LIN {X 0.061,Y -334.260,Z 1455.726,A 0.000,B 0.000,C 90.000,E1 166.589} C_DIS
LIN {X 0.067,Y -335.488,Z 1455.719,A 0.000,B 0.000,C 90.000,E1 165.408} C_DIS
LIN {X 0.143,Y -340.932,Z 1455.695,A 0.000,B 0.000,C 90.000,E1 161.094} C_DIS
LIN {X -0.172,Y -342.138,Z 1455.691,A 0.000,B 0.000,C 90.000,E1 160.369} C_DIS
LIN {X 0.066,Y -342.805,Z 1455.688,A 0.000,B 0.000,C 90.000,E1 159.752} C_DIS
LIN {X 0.060,Y -429.024,Z 1455.688,A 0.000,B 0.000,C 90.000,E1 159.752} C_DIS
LIN {X -0.033,Y -430.016,Z 1455.688,A 0.000,B 0.000,C 90.000,E1 159.752} C_DIS
LIN {X 0.086,Y -433.395,Z 1455.687,A 0.000,B 0.000,C 90.000,E1 159.645} C_DIS
LIN {X -0.050,Y -435.691,Z 1455.687,A 0.000,B 0.000,C 90.000,E1 159.571} C_DIS
LIN {X -0.153,Y -438.470,Z 1455.686,A 0.000,B 0.000,C 90.000,E1 159.444} C_DIS
LIN {X -0.210,Y -444.564,Z 1455.684,A 0.000,B 0.000,C 90.000,E1 159.082} C_DIS
LIN {X 0.199,Y -450.609,Z 1455.681,A 0.000,B 0.000,C 90.000,E1 158.592} C_DIS
LIN {X 0.200,Y -458.142,Z 1455.678,A 0.000,B 0.000,C 90.000,E1 157.975} C_DIS
LIN {X 0.066,Y -470.088,Z 1455.672,A 0.000,B 0.000,C 90.000,E1 156.997} C_DIS
LIN {X 0.090,Y -477.459,Z 1455.669,A 0.000,B 0.000,C 90.000,E1 156.357} C_DIS
LIN {X -0.246,Y -486.291,Z 1455.664,A 0.000,B 0.000,C 90.000,E1 155.613} C_DIS
LIN {X -0.083,Y -496.085,Z 1455.659,A 0.000,B 0.000,C 90.000,E1 154.665} C_DIS
LIN {X -0.227,Y -500.055,Z 1455.657,A 0.000,B 0.000,C 90.000,E1 154.280} C_DIS
LIN {X 0.099,Y -504.054,Z 1455.655,A 0.000,B 0.000,C 90.000,E1 153.819} C_DIS
LIN {X -0.017,Y -509.175,Z 1455.651,A 0.000,B 0.000,C 90.000,E1 153.256} C_DIS
LIN {X -0.087,Y -512.862,Z 1455.649,A 0.000,B 0.000,C 90.000,E1 152.820} C_DIS
LIN {X -0.096,Y -517.315,Z 1455.646,A 0.000,B 0.000,C 90.000,E1 152.231} C_DIS
LIN {X -0.070,Y -521.284,Z 1455.642,A 0.000,B 0.000,C 90.000,E1 151.641} C_DIS
LIN {X -0.011,Y -524.812,Z 1455.639,A 0.000,B 0.000,C 90.000,E1 151.051} C_DIS
LIN {X 0.073,Y -528.055,Z 1455.636,A 0.000,B 0.000,C 90.000,E1 150.461} C_DIS
LIN {X 0.031,Y -531.494,Z 1455.632,A 0.000,B 0.000,C 90.000,E1 149.744} C_DIS
LIN {X 0.289,Y -534.593,Z 1455.628,A 0.000,B 0.000,C 90.000,E1 148.997} C_DIS
LIN {X -0.018,Y -536.856,Z 1455.625,A 0.000,B 0.000,C 90.000,E1 148.456} C_DIS
LIN {X 0.147,Y -538.862,Z 1455.622,A 0.000,B 0.000,C 90.000,E1 147.867} C_DIS
LIN {X -0.121,Y -541.534,Z 1455.617,A 0.000,B 0.000,C 90.000,E1 147.041} C_DIS
LIN {X 0.120,Y -544.822,Z 1455.611,A 0.000,B 0.000,C 90.000,E1 145.881} C_DIS
LIN {X -0.047,Y -547.603,Z 1455.604,A 0.000,B 0.000,C 90.000,E1 144.769} C_DIS
LIN {X 0.044,Y -548.800,Z 1455.601,A 0.000,B 0.000,C 90.000,E1 144.196} C_DIS
LIN {X 0.256,Y -550.997,Z 1455.595,A 0.000,B 0.000,C 90.000,E1 143.050} C_DIS
LIN {X -0.337,Y -552.393,Z 1455.590,A 0.000,B 0.000,C 90.000,E1 142.271} C_DIS
LIN {X 0.198,Y -553.592,Z 1455.586,A 0.000,B 0.000,C 90.000,E1 141.376} C_DIS
LIN {X 0.043,Y -554.950,Z 1455.579,A 0.000,B 0.000,C 90.000,E1 140.275} C_DIS
LIN {X -0.014,Y -556.651,Z 1455.570,A 0.000,B 0.000,C 90.000,E1 138.609} C_DIS
LIN {X -0.047,Y -558.100,Z 1455.561,A 0.000,B 0.000,C 90.000,E1 136.944} C_DIS
LIN {X 0.303,Y -559.361,Z 1455.552,A 0.000,B 0.000,C 90.000,E1 135.243} C_DIS
LIN {X 0.096,Y -559.885,Z 1455.547,A 0.000,B 0.000,C 90.000,E1 134.433} C_DIS
LIN {X 0.020,Y -560.555,Z 1455.539,A 0.000,B 0.000,C 90.000,E1 133.056} C_DIS
LIN {X 0.311,Y -560.929,Z 1455.533,A 0.000,B 0.000,C 90.000,E1 131.919} C_DIS
LIN {X -0.055,Y -561.110,Z 1455.524,A 0.000,B 0.000,C 90.000,E1 130.297} C_DIS
LIN {X -0.264,Y -561.230,Z 1455.513,A 0.000,B 0.000,C 90.000,E1 128.382} C_DIS
LIN {X -0.129,Y -561.256,Z 1455.504,A 0.000,B 0.000,C 90.000,E1 126.710} C_DIS
LIN {X -0.071,Y -561.151,Z 1455.498,A 0.000,B 0.000,C 90.000,E1 125.598} C_DIS
LIN {X 0.087,Y -560.828,Z 1455.490,A 0.000,B 0.000,C 90.000,E1 124.199} C_DIS
LIN {X -0.030,Y -560.379,Z 1455.476,A 0.000,B 0.000,C 90.000,E1 121.720} C_DIS
LIN {X -0.150,Y -560.431,Z 1455.465,A 0.000,B 0.000,C 90.000,E1 119.795} C_DIS
LIN {X -0.046,Y -560.762,Z 1455.455,A 0.000,B 0.000,C 90.000,E1 117.847} C_DIS
LIN {X 0.063,Y -561.275,Z 1455.444,A 0.000,B 0.000,C 90.000,E1 115.899} C_DIS
LIN {X -0.120,Y -561.813,Z 1455.435,A 0.000,B 0.000,C 90.000,E1 114.259} C_DIS
LIN {X -0.314,Y -562.285,Z 1455.427,A 0.000,B 0.000,C 90.000,E1 112.898} C_DIS
LIN {X 0.235,Y -562.746,Z 1455.419,A 0.000,B 0.000,C 90.000,E1 111.461} C_DIS
LIN {X -0.145,Y -563.149,Z 1455.412,A 0.000,B 0.000,C 90.000,E1 110.120} C_DIS
LIN {X 0.255,Y -563.845,Z 1455.400,A 0.000,B 0.000,C 90.000,E1 107.873} C_DIS
LIN {X -0.214,Y -564.772,Z 1455.387,A 0.000,B 0.000,C 90.000,E1 105.717} C_DIS
LIN {X -0.057,Y -564.910,Z 1455.386,A 0.000,B 0.000,C 90.000,E1 105.426} C_DIS
LIN {X 0.027,Y -565.688,Z 1455.381,A 0.000,B 0.000,C 90.000,E1 104.592} C_DIS
LIN {X 0.149,Y -566.655,Z 1455.375,A 0.000,B 0.000,C 90.000,E1 103.480} C_DIS
LIN {X 0.246,Y -567.894,Z 1455.370,A 0.000,B 0.000,C 90.000,E1 102.647} C_DIS
LIN {X -0.133,Y -568.191,Z 1455.369,A 0.000,B 0.000,C 90.000,E1 102.411} C_DIS
LIN {X 0.045,Y -569.125,Z 1455.367,A 0.000,B 0.000,C 90.000,E1 102.119} C_DIS
LIN {X 0.225,Y -569.886,Z 1455.366,A 0.000,B 0.000,C 90.000,E1 101.827} C_DIS
LIN {X 0.036,Y -569.563,Z 1455.363,A 0.000,B 0.000,C 90.000,E1 101.299} C_DIS
LIN {X 0.220,Y -569.627,Z 1455.361,A 0.000,B 0.000,C 90.000,E1 101.007} C_DIS
LIN {X 0.110,Y -569.419,Z 1455.357,A 0.000,B 0.000,C 90.000,E1 100.197} C_DIS
LIN {X -0.083,Y -569.239,Z 1455.354,A 0.000,B 0.000,C 90.000,E1 99.670} C_DIS
LIN {X 0.260,Y -568.151,Z 1455.345,A 0.000,B 0.000,C 90.000,E1 97.992} C_DIS
LIN {X -0.248,Y -568.138,Z 1455.339,A 0.000,B 0.000,C 90.000,E1 96.947} C_DIS
LIN {X -0.202,Y -570.184,Z 1455.319,A 0.000,B 0.000,C 90.000,E1 93.383} C_DIS
LIN {X 0.188,Y -571.720,Z 1455.308,A 0.000,B 0.000,C 90.000,E1 91.432} C_DIS
LIN {X -0.131,Y -573.048,Z 1455.299,A 0.000,B 0.000,C 90.000,E1 89.828} C_DIS
LIN {X 0.005,Y -574.147,Z 1455.292,A 0.000,B 0.000,C 90.000,E1 88.453} C_DIS
LIN {X 0.028,Y -575.123,Z 1455.285,A 0.000,B 0.000,C 90.000,E1 87.364} C_DIS
LIN {X 0.213,Y -576.306,Z 1455.278,A 0.000,B 0.000,C 90.000,E1 85.988} C_DIS
LIN {X 0.222,Y -577.984,Z 1455.267,A 0.000,B 0.000,C 90.000,E1 84.090} C_DIS
LIN {X 0.197,Y -579.406,Z 1455.258,A 0.000,B 0.000,C 90.000,E1 82.470} C_DIS
LIN {X 0.211,Y -580.977,Z 1455.249,A 0.000,B 0.000,C 90.000,E1 80.849} C_DIS
LIN {X -0.222,Y -582.503,Z 1455.240,A 0.000,B 0.000,C 90.000,E1 79.275} C_DIS
LIN {X -0.295,Y -583.830,Z 1455.233,A 0.000,B 0.000,C 90.000,E1 77.937} C_DIS
LIN {X -0.236,Y -585.030,Z 1455.225,A 0.000,B 0.000,C 90.000,E1 76.589} C_DIS
LIN {X 0.222,Y -586.205,Z 1455.216,A 0.000,B 0.000,C 90.000,E1 74.936} C_DIS
LIN {X -0.027,Y -586.651,Z 1455.212,A 0.000,B 0.000,C 90.000,E1 74.157} C_DIS
LIN {X 0.058,Y -587.614,Z 1455.203,A 0.000,B 0.000,C 90.000,E1 72.543} C_DIS
LIN {X -0.083,Y -588.287,Z 1455.196,A 0.000,B 0.000,C 90.000,E1 71.221} C_DIS
LIN {X -0.021,Y -589.004,Z 1455.188,A 0.000,B 0.000,C 90.000,E1 69.880} C_DIS
LIN {X -0.180,Y -590.083,Z 1455.178,A 0.000,B 0.000,C 90.000,E1 68.028} C_DIS
LIN {X 0.026,Y -590.928,Z 1455.169,A 0.000,B 0.000,C 90.000,E1 66.410} C_DIS
LIN {X 0.039,Y -592.327,Z 1455.157,A 0.000,B 0.000,C 90.000,E1 64.280} C_DIS
LIN {X 0.177,Y -593.164,Z 1455.151,A 0.000,B 0.000,C 90.000,E1 63.204} C_DIS
LIN {X -0.300,Y -595.310,Z 1455.135,A 0.000,B 0.000,C 90.000,E1 60.333} C_DIS
LIN {X -0.071,Y -596.270,Z 1455.129,A 0.000,B 0.000,C 90.000,E1 59.253} C_DIS
LIN {X 0.219,Y -597.873,Z 1455.119,A 0.000,B 0.000,C 90.000,E1 57.375} C_DIS
LIN {X 0.026,Y -599.521,Z 1455.109,A 0.000,B 0.000,C 90.000,E1 55.548} C_DIS
LIN {X -0.197,Y -600.841,Z 1455.100,A 0.000,B 0.000,C 90.000,E1 53.989} C_DIS
LIN {X -0.028,Y -601.825,Z 1455.091,A 0.000,B 0.000,C 90.000,E1 52.396} C_DIS
LIN {X -0.087,Y -602.718,Z 1455.084,A 0.000,B 0.000,C 90.000,E1 51.090} C_DIS
LIN {X 0.205,Y -603.243,Z 1455.079,A 0.000,B 0.000,C 90.000,E1 50.275} C_DIS
LIN {X 0.247,Y -603.524,Z 1455.077,A 0.000,B 0.000,C 90.000,E1 49.747} C_DIS
LIN {X 0.135,Y -603.708,Z 1455.069,A 0.000,B 0.000,C 90.000,E1 48.447} C_DIS
LIN {X 0.026,Y -603.994,Z 1455.062,A 0.000,B 0.000,C 90.000,E1 47.148} C_DIS
LIN {X 0.327,Y -604.187,Z 1455.055,A 0.000,B 0.000,C 90.000,E1 45.810} C_DIS
LIN {X -0.036,Y -604.000,Z 1455.049,A 0.000,B 0.000,C 90.000,E1 44.798} C_DIS
LIN {X 0.036,Y -603.534,Z 1455.043,A 0.000,B 0.000,C 90.000,E1 43.743} C_DIS
LIN {X 0.089,Y -602.845,Z 1455.037,A 0.000,B 0.000,C 90.000,E1 42.690} C_DIS
LIN {X -0.076,Y -602.179,Z 1455.033,A 0.000,B 0.000,C 90.000,E1 41.919} C_DIS
LIN {X -0.219,Y -600.878,Z 1455.026,A 0.000,B 0.000,C 90.000,E1 40.620} C_DIS
LIN {X 0.072,Y -599.204,Z 1455.018,A 0.000,B 0.000,C 90.000,E1 39.277} C_DIS
LIN {X -0.042,Y -597.395,Z 1455.011,A 0.000,B 0.000,C 90.000,E1 37.971} C_DIS
LIN {X -0.059,Y -595.733,Z 1455.005,A 0.000,B 0.000,C 90.000,E1 36.916} C_DIS
LIN {X 0.010,Y -593.691,Z 1454.999,A 0.000,B 0.000,C 90.000,E1 35.851} C_DIS
LIN {X 0.318,Y -591.888,Z 1454.995,A 0.000,B 0.000,C 90.000,E1 35.025} C_DIS
LIN {X 0.126,Y -589.909,Z 1454.990,A 0.000,B 0.000,C 90.000,E1 34.246} C_DIS
LIN {X 0.073,Y -587.854,Z 1454.986,A 0.000,B 0.000,C 90.000,E1 33.452} C_DIS
LIN {X -0.166,Y -585.459,Z 1454.981,A 0.000,B 0.000,C 90.000,E1 32.673} C_DIS
LIN {X -0.082,Y -581.947,Z 1454.975,A 0.000,B 0.000,C 90.000,E1 31.592} C_DIS
LIN {X -0.060,Y -579.976,Z 1454.973,A 0.000,B 0.000,C 90.000,E1 31.052} C_DIS
LIN {X -0.201,Y -576.507,Z 1454.968,A 0.000,B 0.000,C 90.000,E1 30.256} C_DIS
LIN {X 0.201,Y -573.334,Z 1454.964,A 0.000,B 0.000,C 90.000,E1 29.539} C_DIS
LIN {X -0.100,Y -568.447,Z 1454.959,A 0.000,B 0.000,C 90.000,E1 28.615} C_DIS
LIN {X 0.221,Y -564.672,Z 1454.955,A 0.000,B 0.000,C 90.000,E1 27.897} C_DIS
LIN {X 0.149,Y -559.808,Z 1454.951,A 0.000,B 0.000,C 90.000,E1 27.078} C_DIS
LIN {X 0.282,Y -554.507,Z 1454.946,A 0.000,B 0.000,C 90.000,E1 26.232} C_DIS
LIN {X -0.158,Y -550.742,Z 1454.943,A 0.000,B 0.000,C 90.000,E1 25.720} C_DIS
LIN {X -0.005,Y -547.790,Z 1454.941,A 0.000,B 0.000,C 90.000,E1 25.283} C_DIS
LIN {X 0.121,Y -540.180,Z 1454.935,A 0.000,B 0.000,C 90.000,E1 24.283} C_DIS
LIN {X -0.054,Y -534.418,Z 1454.931,A 0.000,B 0.000,C 90.000,E1 23.590} C_DIS
LIN {X -0.009,Y -525.864,Z 1454.926,A 0.000,B 0.000,C 90.000,E1 22.589} C_DIS
LIN {X -0.101,Y -520.741,Z 1454.922,A 0.000,B 0.000,C 90.000,E1 22.025} C_DIS
LIN {X -0.243,Y -511.542,Z 1454.917,A 0.000,B 0.000,C 90.000,E1 21.046} C_DIS
LIN {X 0.088,Y -500.576,Z 1454.911,A 0.000,B 0.000,C 90.000,E1 19.885} C_DIS
LIN {X 0.019,Y -492.405,Z 1454.906,A 0.000,B 0.000,C 90.000,E1 19.087} C_DIS
LIN {X 0.151,Y -487.808,Z 1454.904,A 0.000,B 0.000,C 90.000,E1 18.671} C_DIS
LIN {X 0.072,Y -482.816,Z 1454.902,A 0.000,B 0.000,C 90.000,E1 18.308} C_DIS
LIN {X -0.111,Y -479.110,Z 1454.901,A 0.000,B 0.000,C 90.000,E1 18.109} C_DIS
LIN {X -0.157,Y -476.473,Z 1454.900,A 0.000,B 0.000,C 90.000,E1 18.000} C_DIS
LIN {X -0.126,Y -474.326,Z 1454.900,A 0.000,B 0.000,C 90.000,E1 17.946} C_DIS
LIN {X -0.156,Y -473.854,Z 1454.900,A 0.000,B 0.000,C 90.000,E1 17.946} C_DIS
LIN {X -0.147,Y -373.992,Z 1454.900,A 0.000,B 0.000,C 90.000,E1 17.946} C_DIS
LIN {X 0.091,Y -373.673,Z 1454.897,A 0.000,B 0.000,C 90.000,E1 17.528} C_DIS
LIN {X -0.129,Y -368.069,Z 1454.869,A 0.000,B 0.000,C 90.000,E1 12.411} C_DIS
LIN {X 0.039,Y -366.383,Z 1454.854,A 0.000,B 0.000,C 90.000,E1 9.792} C_DIS
LIN {X -0.021,Y -361.732,Z 1454.821,A 0.000,B 0.000,C 90.000,E1 3.841} C_DIS
LIN {X -0.136,Y -360.851,Z 1454.801,A 0.000,B 0.000,C 90.000,E1 0.115} C_DIS
LIN {X -0.053,Y -359.426,Z 1454.770,A 0.000,B 0.000,C 90.000,E1 354.546} C_DIS
LIN {X 0.070,Y -358.890,Z 1454.759,A 0.000,B 0.000,C 90.000,E1 352.648} C_DIS
LIN {X -0.020,Y -359.563,Z 1454.726,A 0.000,B 0.000,C 90.000,E1 346.645} C_DIS
LIN {X 0.001,Y -361.801,Z 1454.684,A 0.000,B 0.000,C 90.000,E1 339.135} C_DIS
LIN {X -0.154,Y -362.053,Z 1454.680,A 0.000,B 0.000,C 90.000,E1 338.411} C_DIS
LIN {X 0.189,Y -365.980,Z 1454.643,A 0.000,B 0.000,C 90.000,E1 331.641} C_DIS
LIN {X 0.029,Y -366.387,Z 1454.639,A 0.000,B 0.000,C 90.000,E1 330.923} C_DIS
LIN {X -0.031,Y -371.355,Z 1454.604,A 0.000,B 0.000,C 90.000,E1 324.642} C_DIS
LIN {X -0.043,Y -371.766,Z 1454.602,A 0.000,B 0.000,C 90.000,E1 324.276} C_DIS
LIN {X 0.013,Y -377.358,Z 1454.567,A 0.000,B 0.000,C 90.000,E1 318.038} C_DIS
LIN {X 0.012,Y -378.235,Z 1454.563,A 0.000,B 0.000,C 90.000,E1 317.310} C_DIS
LIN {X 0.002,Y -383.940,Z 1454.531,A 0.000,B 0.000,C 90.000,E1 311.515} C_DIS
LIN {X 0.088,Y -384.893,Z 1454.527,A 0.000,B 0.000,C 90.000,E1 310.782} C_DIS
LIN {X 0.262,Y -390.610,Z 1454.495,A 0.000,B 0.000,C 90.000,E1 305.025} C_DIS
LIN {X 0.106,Y -391.104,Z 1454.493,A 0.000,B 0.000,C 90.000,E1 304.692} C_DIS
LIN {X 0.022,Y -391.648,Z 1454.489,A 0.000,B 0.000,C 90.000,E1 303.992} C_DIS
LIN {X -0.080,Y -396.825,Z 1454.459,A 0.000,B 0.000,C 90.000,E1 298.693} C_DIS
LIN {X -0.210,Y -397.120,Z 1454.457,A 0.000,B 0.000,C 90.000,E1 298.359} C_DIS
LIN {X -0.055,Y -401.597,Z 1454.426,A 0.000,B 0.000,C 90.000,E1 292.717} C_DIS
LIN {X 0.222,Y -404.659,Z 1454.395,A 0.000,B 0.000,C 90.000,E1 287.094} C_DIS
LIN {X -0.079,Y -404.735,Z 1454.391,A 0.000,B 0.000,C 90.000,E1 286.441} C_DIS
LIN {X 0.214,Y -406.099,Z 1454.364,A 0.000,B 0.000,C 90.000,E1 281.535} C_DIS
LIN {X -0.176,Y -406.094,Z 1454.362,A 0.000,B 0.000,C 90.000,E1 281.243} C_DIS
LIN {X -0.097,Y -405.680,Z 1454.333,A 0.000,B 0.000,C 90.000,E1 276.024} C_DIS
LIN {X -0.165,Y -405.058,Z 1454.328,A 0.000,B 0.000,C 90.000,E1 274.992} C_DIS
LIN {X -0.060,Y -403.497,Z 1454.304,A 0.000,B 0.000,C 90.000,E1 270.802} C_DIS
LIN {X -0.092,Y -403.288,Z 1454.302,A 0.000,B 0.000,C 90.000,E1 270.458} C_DIS
LIN {X 0.091,Y -398.931,Z 1454.271,A 0.000,B 0.000,C 90.000,E1 264.837} C_DIS
LIN {X -0.040,Y -393.108,Z 1454.242,A 0.000,B 0.000,C 90.000,E1 259.567} C_DIS
LIN {X -0.079,Y -392.835,Z 1454.240,A 0.000,B 0.000,C 90.000,E1 259.218} C_DIS
LIN {X 0.034,Y -385.993,Z 1454.212,A 0.000,B 0.000,C 90.000,E1 254.212} C_DIS
LIN {X -0.026,Y -385.267,Z 1454.208,A 0.000,B 0.000,C 90.000,E1 253.504} C_DIS
LIN {X -0.004,Y -384.768,Z 1454.206,A 0.000,B 0.000,C 90.000,E1 253.142} C_DIS
LIN {X 0.221,Y -377.973,Z 1454.182,A 0.000,B 0.000,C 90.000,E1 248.773} C_DIS
LIN {X -0.044,Y -376.233,Z 1454.174,A 0.000,B 0.000,C 90.000,E1 247.358} C_DIS
LIN {X 0.057,Y -374.944,Z 1454.170,A 0.000,B 0.000,C 90.000,E1 246.613} C_DIS
LIN {X -0.208,Y -368.417,Z 1454.148,A 0.000,B 0.000,C 90.000,E1 242.615} C_DIS
LIN {X 0.097,Y -366.047,Z 1454.137,A 0.000,B 0.000,C 90.000,E1 240.717} C_DIS
LIN {X 0.004,Y -359.196,Z 1454.115,A 0.000,B 0.000,C 90.000,E1 236.628} C_DIS
LIN {X 0.021,Y -355.842,Z 1454.100,A 0.000,B 0.000,C 90.000,E1 233.989} C_DIS
LIN {X -0.173,Y -348.793,Z 1454.075,A 0.000,B 0.000,C 90.000,E1 229.461} C_DIS
LIN {X -0.097,Y -346.185,Z 1454.062,A 0.000,B 0.000,C 90.000,E1 227.148} C_DIS
LIN {X -0.088,Y -345.065,Z 1454.058,A 0.000,B 0.000,C 90.000,E1 226.377} C_DIS
LIN {X 0.094,Y -338.586,Z 1454.030,A 0.000,B 0.000,C 90.000,E1 221.310} C_DIS
LIN {X 0.094,Y -336.840,Z 1454.019,A 0.000,B 0.000,C 90.000,E1 219.358} C_DIS
LIN {X 0.014,Y -330.861,Z 1453.988,A 0.000,B 0.000,C 90.000,E1 213.865} C_DIS
LIN {X 0.149,Y -329.296,Z 1453.975,A 0.000,B 0.000,C 90.000,E1 211.465} C_DIS
LIN {X -0.154,Y -324.669,Z 1453.942,A 0.000,B 0.000,C 90.000,E1 205.540} C_DIS
LIN {X 0.174,Y -323.837,Z 1453.928,A 0.000,B 0.000,C 90.000,E1 203.078} C_DIS
LIN {X -0.017,Y -321.124,Z 1453.881,A 0.000,B 0.000,C 90.000,E1 194.662} C_DIS
LIN {X 0.138,Y -320.932,Z 1453.877,A 0.000,B 0.000,C 90.000,E1 193.828} C_DIS
LIN {X -0.076,Y -321.562,Z 1453.832,A 0.000,B 0.000,C 90.000,E1 185.796} C_DIS
LIN {X -0.143,Y -324.415,Z 1453.790,A 0.000,B 0.000,C 90.000,E1 178.165} C_DIS
LIN {X -0.141,Y -325.376,Z 1453.783,A 0.000,B 0.000,C 90.000,E1 176.963} C_DIS
LIN {X -0.100,Y -329.112,Z 1453.750,A 0.000,B 0.000,C 90.000,E1 170.971} C_DIS
LIN {X 0.061,Y -334.260,Z 1453.726,A 0.000,B 0.000,C 90.000,E1 166.589} C_DIS
LIN {X 0.067,Y -335.488,Z 1453.719,A 0.000,B 0.000,C 90.000,E1 165.408} C_DIS
LIN {X 0.143,Y -340.932,Z 1453.695,A 0.000,B 0.000,C 90.000,E1 161.094} C_DIS
LIN {X 0.033,Y -342.089,Z 1453.691,A 0.000,B 0.000,C 90.000,E1 160.369} C_DIS
LIN {X 0.017,Y -422.192,Z 1453.691,A 0.000,B 0.000,C 90.000,E1 160.369} C_DIS
LIN {X -0.214,Y -424.388,Z 1453.691,A 0.000,B 0.000,C 90.000,E1 160.369} C_DIS
LIN {X -0.104,Y -426.356,Z 1453.691,A 0.000,B 0.000,C 90.000,E1 160.296} C_DIS
LIN {X -0.097,Y -429.003,Z 1453.690,A 0.000,B 0.000,C 90.000,E1 160.188} C_DIS
LIN {X -0.214,Y -431.860,Z 1453.689,A 0.000,B 0.000,C 90.000,E1 160.061} C_DIS
LIN {X -0.149,Y -434.914,Z 1453.688,A 0.000,B 0.000,C 90.000,E1 159.880} C_DIS
LIN {X -0.230,Y -437.978,Z 1453.687,A 0.000,B 0.000,C 90.000,E1 159.699} C_DIS
LIN {X 0.171,Y -444.013,Z 1453.685,A 0.000,B 0.000,C 90.000,E1 159.209} C_DIS
LIN {X 0.148,Y -450.072,Z 1453.682,A 0.000,B 0.000,C 90.000,E1 158.720} C_DIS
LIN {X -0.045,Y -465.121,Z 1453.675,A 0.000,B 0.000,C 90.000,E1 157.486} C_DIS
LIN {X -0.224,Y -475.642,Z 1453.670,A 0.000,B 0.000,C 90.000,E1 156.613} C_DIS
LIN {X 0.111,Y -484.431,Z 1453.666,A 0.000,B 0.000,C 90.000,E1 155.793} C_DIS
LIN {X -0.122,Y -491.613,Z 1453.662,A 0.000,B 0.000,C 90.000,E1 155.153} C_DIS
LIN {X 0.108,Y -498.531,Z 1453.658,A 0.000,B 0.000,C 90.000,E1 154.460} C_DIS
LIN {X 0.007,Y -505.152,Z 1453.654,A 0.000,B 0.000,C 90.000,E1 153.768} C_DIS
LIN {X 0.016,Y -509.028,Z 1453.652,A 0.000,B 0.000,C 90.000,E1 153.332} C_DIS
LIN {X 0.016,Y -513.849,Z 1453.649,A 0.000,B 0.000,C 90.000,E1 152.743} C_DIS
LIN {X 0.188,Y -517.252,Z 1453.646,A 0.000,B 0.000,C 90.000,E1 152.281} C_DIS
LIN {X -0.029,Y -521.248,Z 1453.643,A 0.000,B 0.000,C 90.000,E1 151.719} C_DIS
LIN {X -0.133,Y -525.606,Z 1453.639,A 0.000,B 0.000,C 90.000,E1 151.001} C_DIS
LIN {X 0.109,Y -528.058,Z 1453.636,A 0.000,B 0.000,C 90.000,E1 150.539} C_DIS
LIN {X 0.065,Y -531.547,Z 1453.632,A 0.000,B 0.000,C 90.000,E1 149.822} C_DIS
LIN {X -0.138,Y -534.673,Z 1453.628,A 0.000,B 0.000,C 90.000,E1 149.125} C_DIS
LIN {X 0.015,Y -536.937,Z 1453.625,A 0.000,B 0.000,C 90.000,E1 148.535} C_DIS
LIN {X -0.277,Y -538.954,Z 1453.622,A 0.000,B 0.000,C 90.000,E1 147.995} C_DIS
LIN {X -0.090,Y -541.642,Z 1453.617,A 0.000,B 0.000,C 90.000,E1 147.120} C_DIS
LIN {X 0.149,Y -544.927,Z 1453.611,A 0.000,B 0.000,C 90.000,E1 145.960} C_DIS
LIN {X -0.018,Y -547.714,Z 1453.605,A 0.000,B 0.000,C 90.000,E1 144.848} C_DIS
LIN {X 0.071,Y -548.928,Z 1453.602,A 0.000,B 0.000,C 90.000,E1 144.276} C_DIS
LIN {X 0.284,Y -551.125,Z 1453.595,A 0.000,B 0.000,C 90.000,E1 143.130} C_DIS
LIN {X 0.092,Y -552.923,Z 1453.589,A 0.000,B 0.000,C 90.000,E1 142.029} C_DIS
LIN {X 0.293,Y -554.055,Z 1453.584,A 0.000,B 0.000,C 90.000,E1 141.170} C_DIS
LIN {X 0.140,Y -555.357,Z 1453.578,A 0.000,B 0.000,C 90.000,E1 140.070} C_DIS
LIN {X 0.012,Y -556.744,Z 1453.571,A 0.000,B 0.000,C 90.000,E1 138.690} C_DIS
LIN {X -0.018,Y -558.172,Z 1453.561,A 0.000,B 0.000,C 90.000,E1 137.025} C_DIS
LIN {X -0.061,Y -559.419,Z 1453.552,A 0.000,B 0.000,C 90.000,E1 135.364} C_DIS
LIN {X -0.205,Y -560.071,Z 1453.546,A 0.000,B 0.000,C 90.000,E1 134.271} C_DIS
LIN {X 0.131,Y -560.719,Z 1453.538,A 0.000,B 0.000,C 90.000,E1 132.852} C_DIS
LIN {X 0.013,Y -561.021,Z 1453.532,A 0.000,B 0.000,C 90.000,E1 131.757} C_DIS
LIN {X 0.072,Y -561.165,Z 1453.523,A 0.000,B 0.000,C 90.000,E1 130.092} C_DIS
LIN {X -0.130,Y -561.245,Z 1453.512,A 0.000,B 0.000,C 90.000,E1 128.177} C_DIS
LIN {X 0.010,Y -561.246,Z 1453.503,A 0.000,B 0.000,C 90.000,E1 126.503} C_DIS
LIN {X 0.070,Y -561.093,Z 1453.497,A 0.000,B 0.000,C 90.000,E1 125.391} C_DIS
LIN {X 0.134,Y -560.851,Z 1453.491,A 0.000,B 0.000,C 90.000,E1 124.278} C_DIS
LIN {X 0.025,Y -560.386,Z 1453.477,A 0.000,B 0.000,C 90.000,E1 121.799} C_DIS
LIN {X -0.088,Y -560.401,Z 1453.466,A 0.000,B 0.000,C 90.000,E1 119.873} C_DIS
LIN {X 0.284,Y -560.752,Z 1453.455,A 0.000,B 0.000,C 90.000,E1 117.897} C_DIS
LIN {X 0.138,Y -561.251,Z 1453.444,A 0.000,B 0.000,C 90.000,E1 115.976} C_DIS
LIN {X -0.037,Y -561.811,Z 1453.435,A 0.000,B 0.000,C 90.000,E1 114.335} C_DIS
LIN {X -0.006,Y -562.287,Z 1453.427,A 0.000,B 0.000,C 90.000,E1 112.950} C_DIS
LIN {X -0.191,Y -562.759,Z 1453.420,A 0.000,B 0.000,C 90.000,E1 111.589} C_DIS
LIN {X 0.154,Y -563.162,Z 1453.412,A 0.000,B 0.000,C 90.000,E1 110.174} C_DIS
LIN {X 0.155,Y -563.984,Z 1453.398,A 0.000,B 0.000,C 90.000,E1 107.692} C_DIS
LIN {X -0.161,Y -564.613,Z 1453.392,A 0.000,B 0.000,C 90.000,E1 106.622} C_DIS
LIN {X -0.235,Y -565.155,Z 1453.389,A 0.000,B 0.000,C 90.000,E1 106.079} C_DIS
LIN {X 0.236,Y -565.472,Z 1453.386,A 0.000,B 0.000,C 90.000,E1 105.481} C_DIS
LIN {X 0.033,Y -565.836,Z 1453.385,A 0.000,B 0.000,C 90.000,E1 105.300} C_DIS
LIN {X 0.151,Y -566.728,Z 1453.381,A 0.000,B 0.000,C 90.000,E1 104.481} C_DIS
LIN {X 0.108,Y -566.741,Z 1453.381,A 0.000,B 0.000,C 90.000,E1 104.481} C_DIS
LIN {X 0.085,Y -568.453,Z 1453.376,A 0.000,B 0.000,C 90.000,E1 103.647} C_DIS
LIN {X 0.261,Y -568.762,Z 1453.374,A 0.000,B 0.000,C 90.000,E1 103.355} C_DIS
LIN {X 0.253,Y -570.843,Z 1453.370,A 0.000,B 0.000,C 90.000,E1 102.535} C_DIS
LIN {X -0.117,Y -571.767,Z 1453.368,A 0.000,B 0.000,C 90.000,E1 102.299} C_DIS
LIN {X -0.051,Y -572.232,Z 1453.366,A 0.000,B 0.000,C 90.000,E1 101.883} C_DIS
LIN {X 0.267,Y -572.517,Z 1453.365,A 0.000,B 0.000,C 90.000,E1 101.715} C_DIS
LIN {X 0.099,Y -572.809,Z 1453.362,A 0.000,B 0.000,C 90.000,E1 101.186} C_DIS
LIN {X -0.266,Y -572.851,Z 1453.361,A 0.000,B 0.000,C 90.000,E1 100.950} C_DIS
LIN {X -0.070,Y -572.533,Z 1453.359,A 0.000,B 0.000,C 90.000,E1 100.658} C_DIS
LIN {X 0.127,Y -572.455,Z 1453.358,A 0.000,B 0.000,C 90.000,E1 100.366} C_DIS
LIN {X 0.221,Y -571.945,Z 1453.356,A 0.000,B 0.000,C 90.000,E1 100.084} C_DIS
LIN {X 0.047,Y -571.563,Z 1453.353,A 0.000,B 0.000,C 90.000,E1 99.557} C_DIS
LIN {X -0.034,Y -570.180,Z 1453.349,A 0.000,B 0.000,C 90.000,E1 98.746} C_DIS
LIN {X 0.152,Y -569.572,Z 1453.347,A 0.000,B 0.000,C 90.000,E1 98.454} C_DIS
LIN {X 0.104,Y -568.992,Z 1453.345,A 0.000,B 0.000,C 90.000,E1 98.049} C_DIS
LIN {X -0.162,Y -568.709,Z 1453.342,A 0.000,B 0.000,C 90.000,E1 97.530} C_DIS
LIN {X 0.015,Y -568.756,Z 1453.340,A 0.000,B 0.000,C 90.000,E1 97.239} C_DIS
LIN {X -0.271,Y -568.501,Z 1453.337,A 0.000,B 0.000,C 90.000,E1 96.720} C_DIS
LIN {X 0.283,Y -569.347,Z 1453.325,A 0.000,B 0.000,C 90.000,E1 94.473} C_DIS
LIN {X 0.085,Y -570.814,Z 1453.314,A 0.000,B 0.000,C 90.000,E1 92.579} C_DIS
LIN {X -0.240,Y -572.162,Z 1453.305,A 0.000,B 0.000,C 90.000,E1 90.974} C_DIS
LIN {X 0.166,Y -573.729,Z 1453.295,A 0.000,B 0.000,C 90.000,E1 89.026} C_DIS
LIN {X -0.099,Y -575.147,Z 1453.286,A 0.000,B 0.000,C 90.000,E1 87.421} C_DIS
LIN {X 0.273,Y -576.558,Z 1453.277,A 0.000,B 0.000,C 90.000,E1 85.755} C_DIS
LIN {X 0.302,Y -578.263,Z 1453.266,A 0.000,B 0.000,C 90.000,E1 83.856} C_DIS
LIN {X 0.214,Y -579.710,Z 1453.257,A 0.000,B 0.000,C 90.000,E1 82.243} C_DIS
LIN {X 0.092,Y -581.050,Z 1453.250,A 0.000,B 0.000,C 90.000,E1 80.905} C_DIS
LIN {X 0.128,Y -582.583,Z 1453.241,A 0.000,B 0.000,C 90.000,E1 79.285} C_DIS
LIN {X 0.165,Y -583.939,Z 1453.233,A 0.000,B 0.000,C 90.000,E1 77.937} C_DIS
LIN {X 0.227,Y -585.128,Z 1453.226,A 0.000,B 0.000,C 90.000,E1 76.589} C_DIS
LIN {X -0.121,Y -586.121,Z 1453.218,A 0.000,B 0.000,C 90.000,E1 75.283} C_DIS
LIN {X -0.125,Y -586.786,Z 1453.212,A 0.000,B 0.000,C 90.000,E1 74.212} C_DIS
LIN {X -0.033,Y -587.735,Z 1453.203,A 0.000,B 0.000,C 90.000,E1 72.598} C_DIS
LIN {X -0.167,Y -588.408,Z 1453.196,A 0.000,B 0.000,C 90.000,E1 71.275} C_DIS
LIN {X -0.098,Y -589.135,Z 1453.188,A 0.000,B 0.000,C 90.000,E1 69.934} C_DIS
LIN {X 0.079,Y -590.192,Z 1453.178,A 0.000,B 0.000,C 90.000,E1 68.050} C_DIS
LIN {X -0.270,Y -591.053,Z 1453.169,A 0.000,B 0.000,C 90.000,E1 66.485} C_DIS
LIN {X -0.106,Y -592.640,Z 1453.156,A 0.000,B 0.000,C 90.000,E1 64.076} C_DIS
LIN {X 0.042,Y -593.409,Z 1453.150,A 0.000,B 0.000,C 90.000,E1 62.999} C_DIS
LIN {X 0.195,Y -595.442,Z 1453.135,A 0.000,B 0.000,C 90.000,E1 60.333} C_DIS
LIN {X 0.335,Y -596.590,Z 1453.128,A 0.000,B 0.000,C 90.000,E1 58.997} C_DIS
LIN {X -0.105,Y -597.984,Z 1453.119,A 0.000,B 0.000,C 90.000,E1 57.454} C_DIS
LIN {X -0.201,Y -599.385,Z 1453.110,A 0.000,B 0.000,C 90.000,E1 55.881} C_DIS
LIN {X 0.176,Y -600.083,Z 1453.106,A 0.000,B 0.000,C 90.000,E1 55.055} C_DIS
LIN {X -0.280,Y -601.167,Z 1453.099,A 0.000,B 0.000,C 90.000,E1 53.783} C_DIS
LIN {X 0.145,Y -602.380,Z 1453.089,A 0.000,B 0.000,C 90.000,E1 51.904} C_DIS
LIN {X 0.086,Y -603.252,Z 1453.081,A 0.000,B 0.000,C 90.000,E1 50.598} C_DIS
LIN {X 0.169,Y -603.773,Z 1453.075,A 0.000,B 0.000,C 90.000,E1 49.542} C_DIS
LIN {X 0.100,Y -604.075,Z 1453.065,A 0.000,B 0.000,C 90.000,E1 47.715} C_DIS
LIN {X 0.200,Y -604.388,Z 1453.057,A 0.000,B 0.000,C 90.000,E1 46.134} C_DIS
LIN {X 0.267,Y -604.288,Z 1453.051,A 0.000,B 0.000,C 90.000,E1 45.081} C_DIS
LIN {X -0.323,Y -604.032,Z 1453.046,A 0.000,B 0.000,C 90.000,E1 44.352} C_DIS
LIN {X -0.024,Y -603.283,Z 1453.039,A 0.000,B 0.000,C 90.000,E1 43.014} C_DIS
LIN {X 0.016,Y -602.465,Z 1453.033,A 0.000,B 0.000,C 90.000,E1 41.962} C_DIS
LIN {X 0.325,Y -601.194,Z 1453.026,A 0.000,B 0.000,C 90.000,E1 40.620} C_DIS
LIN {X -0.225,Y -599.549,Z 1453.019,A 0.000,B 0.000,C 90.000,E1 39.358} C_DIS
LIN {X 0.038,Y -597.733,Z 1453.011,A 0.000,B 0.000,C 90.000,E1 38.016} C_DIS
LIN {X 0.139,Y -596.110,Z 1453.005,A 0.000,B 0.000,C 90.000,E1 36.950} C_DIS
LIN {X 0.220,Y -594.085,Z 1453.000,A 0.000,B 0.000,C 90.000,E1 35.884} C_DIS
LIN {X 0.270,Y -591.676,Z 1452.994,A 0.000,B 0.000,C 90.000,E1 34.818} C_DIS
LIN {X -0.052,Y -589.005,Z 1452.988,A 0.000,B 0.000,C 90.000,E1 33.785} C_DIS
LIN {X 0.214,Y -586.766,Z 1452.983,A 0.000,B 0.000,C 90.000,E1 32.959} C_DIS
LIN {X -0.177,Y -583.400,Z 1452.977,A 0.000,B 0.000,C 90.000,E1 31.926} C_DIS
LIN {X -0.145,Y -581.551,Z 1452.974,A 0.000,B 0.000,C 90.000,E1 31.386} C_DIS
LIN {X -0.125,Y -579.525,Z 1452.971,A 0.000,B 0.000,C 90.000,E1 30.846} C_DIS
LIN {X 0.302,Y -576.554,Z 1452.968,A 0.000,B 0.000,C 90.000,E1 30.129} C_DIS
LIN {X 0.203,Y -573.396,Z 1452.964,A 0.000,B 0.000,C 90.000,E1 29.461} C_DIS
LIN {X -0.288,Y -569.188,Z 1452.959,A 0.000,B 0.000,C 90.000,E1 28.693} C_DIS
LIN {X -0.046,Y -564.674,Z 1452.955,A 0.000,B 0.000,C 90.000,E1 27.847} C_DIS
LIN {X 0.143,Y -559.815,Z 1452.950,A 0.000,B 0.000,C 90.000,E1 27.001} C_DIS
LIN {X 0.027,Y -554.512,Z 1452.946,A 0.000,B 0.000,C 90.000,E1 26.181} C_DIS
LIN {X 0.211,Y -549.757,Z 1452.942,A 0.000,B 0.000,C 90.000,E1 25.463} C_DIS
LIN {X 0.235,Y -545.611,Z 1452.938,A 0.000,B 0.000,C 90.000,E1 24.899} C_DIS
LIN {X -0.023,Y -539.009,Z 1452.934,A 0.000,B 0.000,C 90.000,E1 24.079} C_DIS
LIN {X -0.072,Y -534.355,Z 1452.931,A 0.000,B 0.000,C 90.000,E1 23.515} C_DIS
LIN {X -0.044,Y -525.756,Z 1452.925,A 0.000,B 0.000,C 90.000,E1 22.514} C_DIS
LIN {X 0.195,Y -519.315,Z 1452.921,A 0.000,B 0.000,C 90.000,E1 21.770} C_DIS
LIN {X 0.249,Y -510.285,Z 1452.916,A 0.000,B 0.000,C 90.000,E1 20.791} C_DIS
LIN {X -0.118,Y -500.840,Z 1452.910,A 0.000,B 0.000,C 90.000,E1 19.866} C_DIS
LIN {X -0.076,Y -490.229,Z 1452.904,A 0.000,B 0.000,C 90.000,E1 18.779} C_DIS
LIN {X -0.098,Y -485.780,Z 1452.902,A 0.000,B 0.000,C 90.000,E1 18.362} C_DIS
LIN {X 0.109,Y -481.112,Z 1452.900,A 0.000,B 0.000,C 90.000,E1 17.946} C_DIS
LIN {X 0.177,Y -477.765,Z 1452.898,A 0.000,B 0.000,C 90.000,E1 17.692} C_DIS
LIN {X -0.172,Y -474.107,Z 1452.897,A 0.000,B 0.000,C 90.000,E1 17.511} C_DIS
LIN {X 0.075,Y -471.106,Z 1452.896,A 0.000,B 0.000,C 90.000,E1 17.347} C_DIS
LIN {X -0.146,Y -469.423,Z 1452.896,A 0.000,B 0.000,C 90.000,E1 17.330} C_DIS
LIN {X 0.235,Y -468.721,Z 1452.896,A 0.000,B 0.000,C 90.000,E1 17.275} C_DIS
LIN {X 0.160,Y -373.384,Z 1452.896,A 0.000,B 0.000,C 90.000,E1 17.275} C_DIS
LIN {X 0.034,Y -367.822,Z 1452.867,A 0.000,B 0.000,C 90.000,E1 12.063} C_DIS
LIN {X -0.020,Y -366.431,Z 1452.855,A 0.000,B 0.000,C 90.000,E1 9.849} C_DIS
LIN {X -0.082,Y -361.753,Z 1452.822,A 0.000,B 0.000,C 90.000,E1 3.898} C_DIS
LIN {X 0.165,Y -360.878,Z 1452.801,A 0.000,B 0.000,C 90.000,E1 0.115} C_DIS
LIN {X -0.053,Y -359.426,Z 1452.770,A 0.000,B 0.000,C 90.000,E1 354.546} C_DIS
LIN {X 0.070,Y -358.890,Z 1452.759,A 0.000,B 0.000,C 90.000,E1 352.648} C_DIS
LIN {X -0.020,Y -359.563,Z 1452.726,A 0.000,B 0.000,C 90.000,E1 346.645} C_DIS
LIN {X 0.001,Y -361.801,Z 1452.684,A 0.000,B 0.000,C 90.000,E1 339.135} C_DIS
LIN {X -0.154,Y -362.053,Z 1452.680,A 0.000,B 0.000,C 90.000,E1 338.411} C_DIS
LIN {X 0.189,Y -365.980,Z 1452.643,A 0.000,B 0.000,C 90.000,E1 331.641} C_DIS
LIN {X 0.029,Y -366.387,Z 1452.639,A 0.000,B 0.000,C 90.000,E1 330.923} C_DIS
LIN {X -0.031,Y -371.355,Z 1452.604,A 0.000,B 0.000,C 90.000,E1 324.642} C_DIS
LIN {X -0.043,Y -371.766,Z 1452.602,A 0.000,B 0.000,C 90.000,E1 324.276} C_DIS
LIN {X 0.013,Y -377.358,Z 1452.567,A 0.000,B 0.000,C 90.000,E1 318.038} C_DIS
LIN {X 0.012,Y -378.235,Z 1452.563,A 0.000,B 0.000,C 90.000,E1 317.310} C_DIS
LIN {X 0.002,Y -383.940,Z 1452.531,A 0.000,B 0.000,C 90.000,E1 311.515} C_DIS
LIN {X 0.088,Y -384.893,Z 1452.527,A 0.000,B 0.000,C 90.000,E1 310.782} C_DIS
LIN {X 0.262,Y -390.610,Z 1452.495,A 0.000,B 0.000,C 90.000,E1 305.025} C_DIS
LIN {X 0.106,Y -391.104,Z 1452.493,A 0.000,B 0.000,C 90.000,E1 304.692} C_DIS
LIN {X 0.022,Y -391.648,Z 1452.489,A 0.000,B 0.000,C 90.000,E1 303.992} C_DIS
LIN {X -0.080,Y -396.825,Z 1452.459,A 0.000,B 0.000,C 90.000,E1 298.693} C_DIS
LIN {X -0.210,Y -397.120,Z 1452.457,A 0.000,B 0.000,C 90.000,E1 298.359} C_DIS
LIN {X -0.055,Y -401.597,Z 1452.426,A 0.000,B 0.000,C 90.000,E1 292.717} C_DIS
LIN {X 0.222,Y -404.659,Z 1452.395,A 0.000,B 0.000,C 90.000,E1 287.094} C_DIS
LIN {X -0.079,Y -404.735,Z 1452.391,A 0.000,B 0.000,C 90.000,E1 286.441} C_DIS
LIN {X 0.214,Y -406.099,Z 1452.364,A 0.000,B 0.000,C 90.000,E1 281.535} C_DIS
LIN {X -0.176,Y -406.094,Z 1452.362,A 0.000,B 0.000,C 90.000,E1 281.243} C_DIS
LIN {X -0.097,Y -405.680,Z 1452.333,A 0.000,B 0.000,C 90.000,E1 276.024} C_DIS
LIN {X -0.165,Y -405.058,Z 1452.328,A 0.000,B 0.000,C 90.000,E1 274.992} C_DIS
LIN {X -0.060,Y -403.497,Z 1452.304,A 0.000,B 0.000,C 90.000,E1 270.802} C_DIS
LIN {X -0.092,Y -403.288,Z 1452.302,A 0.000,B 0.000,C 90.000,E1 270.458} C_DIS
LIN {X 0.091,Y -398.931,Z 1452.271,A 0.000,B 0.000,C 90.000,E1 264.837} C_DIS
LIN {X -0.040,Y -393.108,Z 1452.242,A 0.000,B 0.000,C 90.000,E1 259.567} C_DIS
LIN {X -0.079,Y -392.835,Z 1452.240,A 0.000,B 0.000,C 90.000,E1 259.218} C_DIS
LIN {X 0.034,Y -385.993,Z 1452.212,A 0.000,B 0.000,C 90.000,E1 254.212} C_DIS
LIN {X -0.026,Y -385.267,Z 1452.208,A 0.000,B 0.000,C 90.000,E1 253.504} C_DIS
LIN {X -0.004,Y -384.768,Z 1452.206,A 0.000,B 0.000,C 90.000,E1 253.142} C_DIS
LIN {X 0.221,Y -377.973,Z 1452.182,A 0.000,B 0.000,C 90.000,E1 248.773} C_DIS
LIN {X -0.044,Y -376.233,Z 1452.174,A 0.000,B 0.000,C 90.000,E1 247.358} C_DIS
LIN {X 0.057,Y -374.944,Z 1452.170,A 0.000,B 0.000,C 90.000,E1 246.613} C_DIS
LIN {X -0.208,Y -368.417,Z 1452.148,A 0.000,B 0.000,C 90.000,E1 242.615} C_DIS
LIN {X 0.097,Y -366.047,Z 1452.137,A 0.000,B 0.000,C 90.000,E1 240.717} C_DIS
LIN {X 0.004,Y -359.196,Z 1452.115,A 0.000,B 0.000,C 90.000,E1 236.628} C_DIS
LIN {X 0.021,Y -355.842,Z 1452.100,A 0.000,B 0.000,C 90.000,E1 233.989} C_DIS
LIN {X -0.173,Y -348.793,Z 1452.075,A 0.000,B 0.000,C 90.000,E1 229.461} C_DIS
LIN {X -0.097,Y -346.185,Z 1452.062,A 0.000,B 0.000,C 90.000,E1 227.148} C_DIS
LIN {X -0.088,Y -345.065,Z 1452.058,A 0.000,B 0.000,C 90.000,E1 226.377} C_DIS
LIN {X 0.094,Y -338.586,Z 1452.030,A 0.000,B 0.000,C 90.000,E1 221.310} C_DIS
LIN {X 0.094,Y -336.840,Z 1452.019,A 0.000,B 0.000,C 90.000,E1 219.358} C_DIS
LIN {X 0.014,Y -330.861,Z 1451.988,A 0.000,B 0.000,C 90.000,E1 213.865} C_DIS
LIN {X 0.149,Y -329.296,Z 1451.975,A 0.000,B 0.000,C 90.000,E1 211.465} C_DIS
LIN {X -0.154,Y -324.669,Z 1451.942,A 0.000,B 0.000,C 90.000,E1 205.540} C_DIS
LIN {X 0.174,Y -323.837,Z 1451.928,A 0.000,B 0.000,C 90.000,E1 203.078} C_DIS
LIN {X -0.017,Y -321.124,Z 1451.881,A 0.000,B 0.000,C 90.000,E1 194.662} C_DIS
LIN {X 0.138,Y -320.932,Z 1451.877,A 0.000,B 0.000,C 90.000,E1 193.828} C_DIS
LIN {X -0.076,Y -321.562,Z 1451.832,A 0.000,B 0.000,C 90.000,E1 185.796} C_DIS
LIN {X -0.143,Y -324.415,Z 1451.790,A 0.000,B 0.000,C 90.000,E1 178.165} C_DIS
LIN {X -0.141,Y -325.376,Z 1451.783,A 0.000,B 0.000,C 90.000,E1 176.963} C_DIS
LIN {X -0.100,Y -329.112,Z 1451.750,A 0.000,B 0.000,C 90.000,E1 170.971} C_DIS
LIN {X 0.061,Y -334.260,Z 1451.726,A 0.000,B 0.000,C 90.000,E1 166.589} C_DIS
LIN {X 0.067,Y -335.488,Z 1451.719,A 0.000,B 0.000,C 90.000,E1 165.408} C_DIS
LIN {X 0.160,Y -341.121,Z 1451.694,A 0.000,B 0.000,C 90.000,E1 160.967} C_DIS
LIN {X 0.161,Y -415.832,Z 1451.694,A 0.000,B 0.000,C 90.000,E1 160.967} C_DIS
LIN {X 0.140,Y -418.801,Z 1451.694,A 0.000,B 0.000,C 90.000,E1 160.913} C_DIS
LIN {X 0.117,Y -420.500,Z 1451.694,A 0.000,B 0.000,C 90.000,E1 160.859} C_DIS
LIN {X -0.019,Y -423.825,Z 1451.693,A 0.000,B 0.000,C 90.000,E1 160.732} C_DIS
LIN {X 0.184,Y -426.680,Z 1451.692,A 0.000,B 0.000,C 90.000,E1 160.550} C_DIS
LIN {X -0.022,Y -432.759,Z 1451.690,A 0.000,B 0.000,C 90.000,E1 160.188} C_DIS
LIN {X -0.155,Y -438.952,Z 1451.688,A 0.000,B 0.000,C 90.000,E1 159.752} C_DIS
LIN {X -0.036,Y -449.530,Z 1451.682,A 0.000,B 0.000,C 90.000,E1 158.847} C_DIS
LIN {X 0.231,Y -464.811,Z 1451.675,A 0.000,B 0.000,C 90.000,E1 157.539} C_DIS
LIN {X 0.030,Y -476.769,Z 1451.670,A 0.000,B 0.000,C 90.000,E1 156.538} C_DIS
LIN {X -0.174,Y -485.411,Z 1451.665,A 0.000,B 0.000,C 90.000,E1 155.793} C_DIS
LIN {X 0.056,Y -493.917,Z 1451.661,A 0.000,B 0.000,C 90.000,E1 154.973} C_DIS
LIN {X -0.154,Y -499.373,Z 1451.658,A 0.000,B 0.000,C 90.000,E1 154.460} C_DIS
LIN {X -0.257,Y -505.962,Z 1451.654,A 0.000,B 0.000,C 90.000,E1 153.768} C_DIS
LIN {X 0.015,Y -509.772,Z 1451.652,A 0.000,B 0.000,C 90.000,E1 153.307} C_DIS
LIN {X -0.062,Y -513.426,Z 1451.649,A 0.000,B 0.000,C 90.000,E1 152.871} C_DIS
LIN {X -0.053,Y -517.925,Z 1451.646,A 0.000,B 0.000,C 90.000,E1 152.281} C_DIS
LIN {X -0.018,Y -521.860,Z 1451.643,A 0.000,B 0.000,C 90.000,E1 151.691} C_DIS
LIN {X -0.112,Y -526.185,Z 1451.639,A 0.000,B 0.000,C 90.000,E1 150.973} C_DIS
LIN {X -0.122,Y -528.626,Z 1451.636,A 0.000,B 0.000,C 90.000,E1 150.539} C_DIS
LIN {X 0.105,Y -532.065,Z 1451.632,A 0.000,B 0.000,C 90.000,E1 149.793} C_DIS
LIN {X 0.097,Y -535.172,Z 1451.628,A 0.000,B 0.000,C 90.000,E1 149.076} C_DIS
LIN {X -0.206,Y -537.378,Z 1451.625,A 0.000,B 0.000,C 90.000,E1 148.535} C_DIS
LIN {X -0.039,Y -539.387,Z 1451.622,A 0.000,B 0.000,C 90.000,E1 147.946} C_DIS
LIN {X -0.025,Y -541.246,Z 1451.619,A 0.000,B 0.000,C 90.000,E1 147.375} C_DIS
LIN {X 0.188,Y -543.726,Z 1451.614,A 0.000,B 0.000,C 90.000,E1 146.501} C_DIS
LIN {X -0.029,Y -545.998,Z 1451.609,A 0.000,B 0.000,C 90.000,E1 145.674} C_DIS
LIN {X -0.180,Y -548.715,Z 1451.603,A 0.000,B 0.000,C 90.000,E1 144.562} C_DIS
LIN {X 0.084,Y -551.408,Z 1451.595,A 0.000,B 0.000,C 90.000,E1 143.130} C_DIS
LIN {X -0.105,Y -553.174,Z 1451.589,A 0.000,B 0.000,C 90.000,E1 142.029} C_DIS
LIN {X 0.098,Y -554.281,Z 1451.584,A 0.000,B 0.000,C 90.000,E1 141.170} C_DIS
LIN {X -0.052,Y -555.556,Z 1451.578,A 0.000,B 0.000,C 90.000,E1 140.070} C_DIS
LIN {X -0.176,Y -556.916,Z 1451.570,A 0.000,B 0.000,C 90.000,E1 138.690} C_DIS
LIN {X 0.177,Y -558.307,Z 1451.561,A 0.000,B 0.000,C 90.000,E1 136.986} C_DIS
LIN {X 0.149,Y -559.519,Z 1451.552,A 0.000,B 0.000,C 90.000,E1 135.324} C_DIS
LIN {X 0.003,Y -560.148,Z 1451.546,A 0.000,B 0.000,C 90.000,E1 134.231} C_DIS
LIN {X -0.051,Y -560.772,Z 1451.538,A 0.000,B 0.000,C 90.000,E1 132.852} C_DIS
LIN {X -0.167,Y -561.067,Z 1451.532,A 0.000,B 0.000,C 90.000,E1 131.757} C_DIS
LIN {X -0.108,Y -561.165,Z 1451.523,A 0.000,B 0.000,C 90.000,E1 130.092} C_DIS
LIN {X 0.034,Y -561.259,Z 1451.514,A 0.000,B 0.000,C 90.000,E1 128.418} C_DIS
LIN {X 0.183,Y -561.249,Z 1451.504,A 0.000,B 0.000,C 90.000,E1 126.744} C_DIS
LIN {X 0.120,Y -561.118,Z 1451.498,A 0.000,B 0.000,C 90.000,E1 125.644} C_DIS
LIN {X -0.045,Y -560.846,Z 1451.490,A 0.000,B 0.000,C 90.000,E1 124.278} C_DIS
LIN {X -0.238,Y -560.411,Z 1451.478,A 0.000,B 0.000,C 90.000,E1 122.084} C_DIS
LIN {X 0.146,Y -560.361,Z 1451.469,A 0.000,B 0.000,C 90.000,E1 120.384} C_DIS
LIN {X 0.104,Y -560.770,Z 1451.455,A 0.000,B 0.000,C 90.000,E1 117.897} C_DIS
LIN {X -0.041,Y -561.285,Z 1451.444,A 0.000,B 0.000,C 90.000,E1 115.976} C_DIS
LIN {X -0.216,Y -561.842,Z 1451.435,A 0.000,B 0.000,C 90.000,E1 114.335} C_DIS
LIN {X -0.185,Y -562.317,Z 1451.427,A 0.000,B 0.000,C 90.000,E1 112.950} C_DIS
LIN {X 0.154,Y -562.790,Z 1451.420,A 0.000,B 0.000,C 90.000,E1 111.535} C_DIS
LIN {X 0.104,Y -563.256,Z 1451.411,A 0.000,B 0.000,C 90.000,E1 109.885} C_DIS
LIN {X -0.022,Y -564.148,Z 1451.398,A 0.000,B 0.000,C 90.000,E1 107.692} C_DIS
LIN {X 0.125,Y -564.278,Z 1451.397,A 0.000,B 0.000,C 90.000,E1 107.402} C_DIS
LIN {X 0.273,Y -565.644,Z 1451.390,A 0.000,B 0.000,C 90.000,E1 106.079} C_DIS
LIN {X 0.305,Y -566.919,Z 1451.387,A 0.000,B 0.000,C 90.000,E1 105.662} C_DIS
LIN {X -0.192,Y -567.577,Z 1451.385,A 0.000,B 0.000,C 90.000,E1 105.300} C_DIS
LIN {X 0.092,Y -568.306,Z 1451.384,A 0.000,B 0.000,C 90.000,E1 105.134} C_DIS
LIN {X -0.138,Y -569.350,Z 1451.383,A 0.000,B 0.000,C 90.000,E1 104.883} C_DIS
LIN {X 0.151,Y -569.717,Z 1451.382,A 0.000,B 0.000,C 90.000,E1 104.717} C_DIS
LIN {X 0.036,Y -570.247,Z 1451.381,A 0.000,B 0.000,C 90.000,E1 104.592} C_DIS
LIN {X 0.255,Y -572.317,Z 1451.379,A 0.000,B 0.000,C 90.000,E1 104.245} C_DIS
LIN {X 0.140,Y -572.933,Z 1451.379,A 0.000,B 0.000,C 90.000,E1 104.120} C_DIS
LIN {X -0.029,Y -574.870,Z 1451.375,A 0.000,B 0.000,C 90.000,E1 103.592} C_DIS
LIN {X -0.184,Y -576.383,Z 1451.373,A 0.000,B 0.000,C 90.000,E1 103.063} C_DIS
LIN {X 0.024,Y -577.091,Z 1451.371,A 0.000,B 0.000,C 90.000,E1 102.771} C_DIS
LIN {X -0.113,Y -578.167,Z 1451.368,A 0.000,B 0.000,C 90.000,E1 102.243} C_DIS
LIN {X -0.243,Y -578.777,Z 1451.365,A 0.000,B 0.000,C 90.000,E1 101.715} C_DIS
LIN {X -0.023,Y -578.969,Z 1451.364,A 0.000,B 0.000,C 90.000,E1 101.422} C_DIS
LIN {X 0.198,Y -578.822,Z 1451.362,A 0.000,B 0.000,C 90.000,E1 101.130} C_DIS
LIN {X -0.149,Y -578.843,Z 1451.360,A 0.000,B 0.000,C 90.000,E1 100.894} C_DIS
LIN {X 0.292,Y -577.924,Z 1451.358,A 0.000,B 0.000,C 90.000,E1 100.310} C_DIS
LIN {X -0.297,Y -575.962,Z 1451.353,A 0.000,B 0.000,C 90.000,E1 99.557} C_DIS
LIN {X -0.086,Y -575.114,Z 1451.351,A 0.000,B 0.000,C 90.000,E1 99.265} C_DIS
LIN {X 0.120,Y -574.087,Z 1451.350,A 0.000,B 0.000,C 90.000,E1 98.973} C_DIS
LIN {X 0.236,Y -572.848,Z 1451.349,A 0.000,B 0.000,C 90.000,E1 98.690} C_DIS
LIN {X 0.032,Y -572.074,Z 1451.347,A 0.000,B 0.000,C 90.000,E1 98.454} C_DIS
LIN {X 0.272,Y -571.791,Z 1451.346,A 0.000,B 0.000,C 90.000,E1 98.276} C_DIS
LIN {X -0.184,Y -571.062,Z 1451.345,A 0.000,B 0.000,C 90.000,E1 98.049} C_DIS
LIN {X 0.228,Y -570.160,Z 1451.342,A 0.000,B 0.000,C 90.000,E1 97.473} C_DIS
LIN {X 0.183,Y -569.245,Z 1451.339,A 0.000,B 0.000,C 90.000,E1 97.068} C_DIS
LIN {X -0.260,Y -568.915,Z 1451.336,A 0.000,B 0.000,C 90.000,E1 96.429} C_DIS
LIN {X -0.152,Y -569.120,Z 1451.328,A 0.000,B 0.000,C 90.000,E1 95.049} C_DIS
LIN {X 0.062,Y -571.030,Z 1451.313,A 0.000,B 0.000,C 90.000,E1 92.293} C_DIS
LIN {X -0.256,Y -572.412,Z 1451.304,A 0.000,B 0.000,C 90.000,E1 90.688} C_DIS
LIN {X 0.014,Y -573.776,Z 1451.295,A 0.000,B 0.000,C 90.000,E1 89.026} C_DIS
LIN {X -0.251,Y -575.193,Z 1451.286,A 0.000,B 0.000,C 90.000,E1 87.421} C_DIS
LIN {X -0.065,Y -576.413,Z 1451.278,A 0.000,B 0.000,C 90.000,E1 86.045} C_DIS
LIN {X 0.152,Y -578.367,Z 1451.266,A 0.000,B 0.000,C 90.000,E1 83.856} C_DIS
LIN {X 0.066,Y -579.819,Z 1451.257,A 0.000,B 0.000,C 90.000,E1 82.243} C_DIS
LIN {X -0.054,Y -581.158,Z 1451.250,A 0.000,B 0.000,C 90.000,E1 80.905} C_DIS
LIN {X -0.016,Y -582.723,Z 1451.240,A 0.000,B 0.000,C 90.000,E1 79.285} C_DIS
LIN {X 0.262,Y -584.323,Z 1451.232,A 0.000,B 0.000,C 90.000,E1 77.645} C_DIS
LIN {X -0.241,Y -585.459,Z 1451.224,A 0.000,B 0.000,C 90.000,E1 76.353} C_DIS
LIN {X 0.226,Y -586.637,Z 1451.215,A 0.000,B 0.000,C 90.000,E1 74.700} C_DIS
LIN {X -0.167,Y -587.890,Z 1451.203,A 0.000,B 0.000,C 90.000,E1 72.598} C_DIS
LIN {X 0.026,Y -588.423,Z 1451.197,A 0.000,B 0.000,C 90.000,E1 71.511} C_DIS
LIN {X -0.101,Y -589.153,Z 1451.190,A 0.000,B 0.000,C 90.000,E1 70.188} C_DIS
LIN {X 0.173,Y -590.318,Z 1451.178,A 0.000,B 0.000,C 90.000,E1 68.028} C_DIS
LIN {X 0.149,Y -591.213,Z 1451.169,A 0.000,B 0.000,C 90.000,E1 66.433} C_DIS
LIN {X 0.211,Y -592.986,Z 1451.154,A 0.000,B 0.000,C 90.000,E1 63.768} C_DIS
LIN {X -0.077,Y -593.531,Z 1451.150,A 0.000,B 0.000,C 90.000,E1 62.999} C_DIS
LIN {X 0.163,Y -594.661,Z 1451.141,A 0.000,B 0.000,C 90.000,E1 61.385} C_DIS
LIN {X -0.011,Y -595.812,Z 1451.134,A 0.000,B 0.000,C 90.000,E1 60.078} C_DIS
LIN {X 0.225,Y -596.756,Z 1451.128,A 0.000,B 0.000,C 90.000,E1 58.997} C_DIS
LIN {X 0.017,Y -598.382,Z 1451.118,A 0.000,B 0.000,C 90.000,E1 57.168} C_DIS
LIN {X 0.175,Y -600.054,Z 1451.107,A 0.000,B 0.000,C 90.000,E1 55.308} C_DIS
LIN {X 0.213,Y -601.149,Z 1451.100,A 0.000,B 0.000,C 90.000,E1 53.989} C_DIS
LIN {X 0.023,Y -602.189,Z 1451.091,A 0.000,B 0.000,C 90.000,E1 52.431} C_DIS
LIN {X 0.083,Y -602.889,Z 1451.086,A 0.000,B 0.000,C 90.000,E1 51.376} C_DIS
LIN {X -0.219,Y -603.559,Z 1451.080,A 0.000,B 0.000,C 90.000,E1 50.356} C_DIS
LIN {X 0.079,Y -603.938,Z 1451.075,A 0.000,B 0.000,C 90.000,E1 49.542} C_DIS
LIN {X 0.171,Y -604.077,Z 1451.069,A 0.000,B 0.000,C 90.000,E1 48.485} C_DIS
LIN {X -0.141,Y -604.417,Z 1451.061,A 0.000,B 0.000,C 90.000,E1 46.944} C_DIS
LIN {X -0.079,Y -604.576,Z 1451.055,A 0.000,B 0.000,C 90.000,E1 45.891} C_DIS
LIN {X -0.008,Y -604.403,Z 1451.049,A 0.000,B 0.000,C 90.000,E1 44.838} C_DIS
LIN {X 0.060,Y -603.959,Z 1451.043,A 0.000,B 0.000,C 90.000,E1 43.785} C_DIS
LIN {X -0.297,Y -603.263,Z 1451.037,A 0.000,B 0.000,C 90.000,E1 42.771} C_DIS
LIN {X 0.187,Y -602.428,Z 1451.032,A 0.000,B 0.000,C 90.000,E1 41.676} C_DIS
LIN {X 0.258,Y -601.416,Z 1451.026,A 0.000,B 0.000,C 90.000,E1 40.620} C_DIS
LIN {X 0.092,Y -599.815,Z 1451.019,A 0.000,B 0.000,C 90.000,E1 39.322} C_DIS
LIN {X -0.021,Y -597.998,Z 1451.011,A 0.000,B 0.000,C 90.000,E1 38.016} C_DIS
LIN {X 0.084,Y -596.390,Z 1451.005,A 0.000,B 0.000,C 90.000,E1 36.950} C_DIS
LIN {X 0.067,Y -595.427,Z 1451.002,A 0.000,B 0.000,C 90.000,E1 36.423} C_DIS
LIN {X -0.213,Y -593.207,Z 1450.997,A 0.000,B 0.000,C 90.000,E1 35.391} C_DIS
LIN {X -0.176,Y -590.643,Z 1450.991,A 0.000,B 0.000,C 90.000,E1 34.326} C_DIS
LIN {X 0.106,Y -588.613,Z 1450.986,A 0.000,B 0.000,C 90.000,E1 33.499} C_DIS
LIN {X 0.047,Y -586.280,Z 1450.982,A 0.000,B 0.000,C 90.000,E1 32.704} C_DIS
LIN {X -0.213,Y -583.772,Z 1450.977,A 0.000,B 0.000,C 90.000,E1 31.926} C_DIS
LIN {X -0.177,Y -581.930,Z 1450.974,A 0.000,B 0.000,C 90.000,E1 31.386} C_DIS
LIN {X -0.155,Y -579.902,Z 1450.971,A 0.000,B 0.000,C 90.000,E1 30.846} C_DIS
LIN {X 0.276,Y -576.964,Z 1450.968,A 0.000,B 0.000,C 90.000,E1 30.129} C_DIS
LIN {X 0.018,Y -572.482,Z 1450.962,A 0.000,B 0.000,C 90.000,E1 29.205} C_DIS
LIN {X 0.117,Y -566.656,Z 1450.956,A 0.000,B 0.000,C 90.000,E1 28.103} C_DIS
LIN {X 0.326,Y -561.915,Z 1450.952,A 0.000,B 0.000,C 90.000,E1 27.257} C_DIS
LIN {X -0.168,Y -557.711,Z 1450.948,A 0.000,B 0.000,C 90.000,E1 26.616} C_DIS
LIN {X -0.062,Y -552.245,Z 1450.943,A 0.000,B 0.000,C 90.000,E1 25.771} C_DIS
LIN {X -0.021,Y -548.308,Z 1450.940,A 0.000,B 0.000,C 90.000,E1 25.207} C_DIS
LIN {X -0.129,Y -542.934,Z 1450.936,A 0.000,B 0.000,C 90.000,E1 24.515} C_DIS
LIN {X 0.208,Y -537.300,Z 1450.932,A 0.000,B 0.000,C 90.000,E1 23.770} C_DIS
LIN {X 0.003,Y -531.301,Z 1450.928,A 0.000,B 0.000,C 90.000,E1 23.078} C_DIS
LIN {X 0.074,Y -523.729,Z 1450.923,A 0.000,B 0.000,C 90.000,E1 22.206} C_DIS
LIN {X 0.154,Y -517.270,Z 1450.919,A 0.000,B 0.000,C 90.000,E1 21.482} C_DIS
LIN {X 0.312,Y -508.063,Z 1450.914,A 0.000,B 0.000,C 90.000,E1 20.482} C_DIS
LIN {X -0.114,Y -499.724,Z 1450.909,A 0.000,B 0.000,C 90.000,E1 19.685} C_DIS
LIN {X -0.139,Y -486.143,Z 1450.902,A 0.000,B 0.000,C 90.000,E1 18.290} C_DIS
LIN {X -0.204,Y -481.793,Z 1450.899,A 0.000,B 0.000,C 90.000,E1 17.873} C_DIS
LIN {X -0.114,Y -477.149,Z 1450.897,A 0.000,B 0.000,C 90.000,E1 17.457} C_DIS
LIN {X -0.201,Y -472.255,Z 1450.895,A 0.000,B 0.000,C 90.000,E1 17.094} C_DIS
LIN {X -0.119,Y -468.611,Z 1450.894,A 0.000,B 0.000,C 90.000,E1 16.858} C_DIS
LIN {X 0.243,Y -465.445,Z 1450.893,A 0.000,B 0.000,C 90.000,E1 16.677} C_DIS
LIN {X -0.038,Y -463.904,Z 1450.893,A 0.000,B 0.000,C 90.000,E1 16.677} C_DIS
LIN {X -0.078,Y -463.215,Z 1450.893,A 0.000,B 0.000,C 90.000,E1 16.677} C_DIS
LIN {X -0.095,Y -372.527,Z 1450.893,A 0.000,B 0.000,C 90.000,E1 16.677} C_DIS
LIN {X -0.042,Y -367.359,Z 1450.864,A 0.000,B 0.000,C 90.000,E1 11.422} C_DIS
LIN {X -0.179,Y -366.491,Z 1450.855,A 0.000,B 0.000,C 90.000,E1 9.962} C_DIS
LIN {X 0.117,Y -361.793,Z 1450.822,A 0.000,B 0.000,C 90.000,E1 3.955} C_DIS
LIN {X 0.003,Y -360.903,Z 1450.801,A 0.000,B 0.000,C 90.000,E1 0.229} C_DIS
LIN {X -0.053,Y -359.426,Z 1450.770,A 0.000,B 0.000,C 90.000,E1 354.546} C_DIS
LIN {X 0.070,Y -358.890,Z 1450.759,A 0.000,B 0.000,C 90.000,E1 352.648} C_DIS
LIN {X -0.020,Y -359.563,Z 1450.726,A 0.000,B 0.000,C 90.000,E1 346.645} C_DIS
LIN {X 0.001,Y -361.801,Z 1450.684,A 0.000,B 0.000,C 90.000,E1 339.135} C_DIS
LIN {X -0.154,Y -362.053,Z 1450.680,A 0.000,B 0.000,C 90.000,E1 338.411} C_DIS
LIN {X 0.189,Y -365.980,Z 1450.643,A 0.000,B 0.000,C 90.000,E1 331.641} C_DIS
LIN {X 0.029,Y -366.387,Z 1450.639,A 0.000,B 0.000,C 90.000,E1 330.923} C_DIS
LIN {X -0.031,Y -371.355,Z 1450.604,A 0.000,B 0.000,C 90.000,E1 324.642} C_DIS
LIN {X -0.043,Y -371.766,Z 1450.602,A 0.000,B 0.000,C 90.000,E1 324.276} C_DIS
LIN {X 0.013,Y -377.358,Z 1450.567,A 0.000,B 0.000,C 90.000,E1 318.038} C_DIS
LIN {X 0.012,Y -378.235,Z 1450.563,A 0.000,B 0.000,C 90.000,E1 317.310} C_DIS
LIN {X 0.002,Y -383.940,Z 1450.531,A 0.000,B 0.000,C 90.000,E1 311.515} C_DIS
LIN {X 0.088,Y -384.893,Z 1450.527,A 0.000,B 0.000,C 90.000,E1 310.782} C_DIS
LIN {X 0.262,Y -390.610,Z 1450.495,A 0.000,B 0.000,C 90.000,E1 305.025} C_DIS
LIN {X 0.106,Y -391.104,Z 1450.493,A 0.000,B 0.000,C 90.000,E1 304.692} C_DIS
LIN {X 0.022,Y -391.648,Z 1450.489,A 0.000,B 0.000,C 90.000,E1 303.992} C_DIS
LIN {X -0.080,Y -396.825,Z 1450.459,A 0.000,B 0.000,C 90.000,E1 298.693} C_DIS
LIN {X -0.210,Y -397.120,Z 1450.457,A 0.000,B 0.000,C 90.000,E1 298.359} C_DIS
LIN {X -0.055,Y -401.597,Z 1450.426,A 0.000,B 0.000,C 90.000,E1 292.717} C_DIS
LIN {X 0.222,Y -404.659,Z 1450.395,A 0.000,B 0.000,C 90.000,E1 287.094} C_DIS
LIN {X -0.079,Y -404.735,Z 1450.391,A 0.000,B 0.000,C 90.000,E1 286.441} C_DIS
LIN {X 0.214,Y -406.099,Z 1450.364,A 0.000,B 0.000,C 90.000,E1 281.535} C_DIS
LIN {X -0.176,Y -406.094,Z 1450.362,A 0.000,B 0.000,C 90.000,E1 281.243} C_DIS
LIN {X -0.097,Y -405.680,Z 1450.333,A 0.000,B 0.000,C 90.000,E1 276.024} C_DIS
LIN {X -0.165,Y -405.058,Z 1450.328,A 0.000,B 0.000,C 90.000,E1 274.992} C_DIS
LIN {X -0.060,Y -403.497,Z 1450.304,A 0.000,B 0.000,C 90.000,E1 270.802} C_DIS
LIN {X -0.092,Y -403.288,Z 1450.302,A 0.000,B 0.000,C 90.000,E1 270.458} C_DIS
LIN {X 0.091,Y -398.931,Z 1450.271,A 0.000,B 0.000,C 90.000,E1 264.837} C_DIS
LIN {X -0.040,Y -393.108,Z 1450.242,A 0.000,B 0.000,C 90.000,E1 259.567} C_DIS
LIN {X -0.079,Y -392.835,Z 1450.240,A 0.000,B 0.000,C 90.000,E1 259.218} C_DIS
LIN {X 0.034,Y -385.993,Z 1450.212,A 0.000,B 0.000,C 90.000,E1 254.212} C_DIS
LIN {X -0.026,Y -385.267,Z 1450.208,A 0.000,B 0.000,C 90.000,E1 253.504} C_DIS
LIN {X -0.004,Y -384.768,Z 1450.206,A 0.000,B 0.000,C 90.000,E1 253.142} C_DIS
LIN {X 0.221,Y -377.973,Z 1450.182,A 0.000,B 0.000,C 90.000,E1 248.773} C_DIS
LIN {X -0.044,Y -376.233,Z 1450.174,A 0.000,B 0.000,C 90.000,E1 247.358} C_DIS
LIN {X 0.057,Y -374.944,Z 1450.170,A 0.000,B 0.000,C 90.000,E1 246.613} C_DIS
LIN {X -0.208,Y -368.417,Z 1450.148,A 0.000,B 0.000,C 90.000,E1 242.615} C_DIS
LIN {X 0.097,Y -366.047,Z 1450.137,A 0.000,B 0.000,C 90.000,E1 240.717} C_DIS
LIN {X 0.004,Y -359.196,Z 1450.115,A 0.000,B 0.000,C 90.000,E1 236.628} C_DIS
LIN {X 0.021,Y -355.842,Z 1450.100,A 0.000,B 0.000,C 90.000,E1 233.989} C_DIS
LIN {X -0.173,Y -348.793,Z 1450.075,A 0.000,B 0.000,C 90.000,E1 229.461} C_DIS
LIN {X -0.097,Y -346.185,Z 1450.062,A 0.000,B 0.000,C 90.000,E1 227.148} C_DIS
LIN {X -0.088,Y -345.065,Z 1450.058,A 0.000,B 0.000,C 90.000,E1 226.377} C_DIS
LIN {X 0.094,Y -338.586,Z 1450.030,A 0.000,B 0.000,C 90.000,E1 221.310} C_DIS
LIN {X 0.094,Y -336.840,Z 1450.019,A 0.000,B 0.000,C 90.000,E1 219.358} C_DIS
LIN {X 0.014,Y -330.861,Z 1449.988,A 0.000,B 0.000,C 90.000,E1 213.865} C_DIS
LIN {X 0.149,Y -329.296,Z 1449.975,A 0.000,B 0.000,C 90.000,E1 211.465} C_DIS
LIN {X -0.154,Y -324.669,Z 1449.942,A 0.000,B 0.000,C 90.000,E1 205.540} C_DIS
LIN {X 0.174,Y -323.837,Z 1449.928,A 0.000,B 0.000,C 90.000,E1 203.078} C_DIS
LIN {X -0.017,Y -321.124,Z 1449.881,A 0.000,B 0.000,C 90.000,E1 194.662} C_DIS
LIN {X 0.138,Y -320.932,Z 1449.877,A 0.000,B 0.000,C 90.000,E1 193.828} C_DIS
LIN {X -0.076,Y -321.562,Z 1449.832,A 0.000,B 0.000,C 90.000,E1 185.796} C_DIS
LIN {X -0.143,Y -324.415,Z 1449.790,A 0.000,B 0.000,C 90.000,E1 178.165} C_DIS
LIN {X -0.141,Y -325.376,Z 1449.783,A 0.000,B 0.000,C 90.000,E1 176.963} C_DIS
LIN {X -0.100,Y -329.112,Z 1449.750,A 0.000,B 0.000,C 90.000,E1 170.971} C_DIS
LIN {X 0.061,Y -334.260,Z 1449.726,A 0.000,B 0.000,C 90.000,E1 166.589} C_DIS
LIN {X 0.067,Y -335.488,Z 1449.719,A 0.000,B 0.000,C 90.000,E1 165.408} C_DIS
LIN {X -0.059,Y -340.174,Z 1449.698,A 0.000,B 0.000,C 90.000,E1 161.638} C_DIS
LIN {X -0.109,Y -408.763,Z 1449.698,A 0.000,B 0.000,C 90.000,E1 161.638} C_DIS
LIN {X -0.132,Y -412.079,Z 1449.698,A 0.000,B 0.000,C 90.000,E1 161.583} C_DIS
LIN {X -0.026,Y -413.762,Z 1449.697,A 0.000,B 0.000,C 90.000,E1 161.511} C_DIS
LIN {X -0.127,Y -416.576,Z 1449.697,A 0.000,B 0.000,C 90.000,E1 161.402} C_DIS
LIN {X 0.077,Y -419.505,Z 1449.696,A 0.000,B 0.000,C 90.000,E1 161.221} C_DIS
LIN {X 0.084,Y -422.533,Z 1449.695,A 0.000,B 0.000,C 90.000,E1 161.040} C_DIS
LIN {X -0.066,Y -425.607,Z 1449.694,A 0.000,B 0.000,C 90.000,E1 160.859} C_DIS
LIN {X -0.182,Y -431.683,Z 1449.691,A 0.000,B 0.000,C 90.000,E1 160.423} C_DIS
LIN {X 0.099,Y -439.407,Z 1449.688,A 0.000,B 0.000,C 90.000,E1 159.752} C_DIS
LIN {X 0.099,Y -454.576,Z 1449.680,A 0.000,B 0.000,C 90.000,E1 158.465} C_DIS
LIN {X -0.059,Y -465.313,Z 1449.676,A 0.000,B 0.000,C 90.000,E1 157.592} C_DIS
LIN {X 0.130,Y -477.261,Z 1449.670,A 0.000,B 0.000,C 90.000,E1 156.538} C_DIS
LIN {X -0.169,Y -484.593,Z 1449.666,A 0.000,B 0.000,C 90.000,E1 155.921} C_DIS
LIN {X 0.000,Y -493.266,Z 1449.662,A 0.000,B 0.000,C 90.000,E1 155.101} C_DIS
LIN {X 0.168,Y -498.850,Z 1449.659,A 0.000,B 0.000,C 90.000,E1 154.537} C_DIS
LIN {X 0.075,Y -505.462,Z 1449.655,A 0.000,B 0.000,C 90.000,E1 153.845} C_DIS
LIN {X -0.142,Y -509.381,Z 1449.652,A 0.000,B 0.000,C 90.000,E1 153.435} C_DIS
LIN {X 0.102,Y -514.171,Z 1449.649,A 0.000,B 0.000,C 90.000,E1 152.820} C_DIS
LIN {X -0.185,Y -517.626,Z 1449.647,A 0.000,B 0.000,C 90.000,E1 152.410} C_DIS
LIN {X 0.305,Y -521.605,Z 1449.643,A 0.000,B 0.000,C 90.000,E1 151.769} C_DIS
LIN {X 0.210,Y -525.992,Z 1449.639,A 0.000,B 0.000,C 90.000,E1 151.051} C_DIS
LIN {X 0.305,Y -529.201,Z 1449.636,A 0.000,B 0.000,C 90.000,E1 150.461} C_DIS
LIN {X -0.186,Y -532.614,Z 1449.632,A 0.000,B 0.000,C 90.000,E1 149.793} C_DIS
LIN {X -0.045,Y -535.122,Z 1449.629,A 0.000,B 0.000,C 90.000,E1 149.203} C_DIS
LIN {X 0.111,Y -537.344,Z 1449.626,A 0.000,B 0.000,C 90.000,E1 148.614} C_DIS
LIN {X -0.177,Y -540.301,Z 1449.621,A 0.000,B 0.000,C 90.000,E1 147.788} C_DIS
LIN {X 0.009,Y -542.139,Z 1449.618,A 0.000,B 0.000,C 90.000,E1 147.199} C_DIS
LIN {X 0.075,Y -544.519,Z 1449.613,A 0.000,B 0.000,C 90.000,E1 146.342} C_DIS
LIN {X -0.089,Y -547.433,Z 1449.607,A 0.000,B 0.000,C 90.000,E1 145.229} C_DIS
LIN {X -0.315,Y -548.773,Z 1449.604,A 0.000,B 0.000,C 90.000,E1 144.689} C_DIS
LIN {X -0.104,Y -550.933,Z 1449.597,A 0.000,B 0.000,C 90.000,E1 143.543} C_DIS
LIN {X 0.078,Y -552.364,Z 1449.593,A 0.000,B 0.000,C 90.000,E1 142.683} C_DIS
LIN {X 0.342,Y -554.020,Z 1449.587,A 0.000,B 0.000,C 90.000,E1 141.537} C_DIS
LIN {X -0.166,Y -555.632,Z 1449.579,A 0.000,B 0.000,C 90.000,E1 140.194} C_DIS
LIN {X 0.137,Y -556.960,Z 1449.571,A 0.000,B 0.000,C 90.000,E1 138.771} C_DIS
LIN {X 0.040,Y -558.110,Z 1449.563,A 0.000,B 0.000,C 90.000,E1 137.391} C_DIS
LIN {X 0.341,Y -559.159,Z 1449.556,A 0.000,B 0.000,C 90.000,E1 135.972} C_DIS
LIN {X 0.131,Y -559.700,Z 1449.551,A 0.000,B 0.000,C 90.000,E1 135.162} C_DIS
LIN {X -0.073,Y -560.166,Z 1449.546,A 0.000,B 0.000,C 90.000,E1 134.352} C_DIS
LIN {X 0.266,Y -560.759,Z 1449.539,A 0.000,B 0.000,C 90.000,E1 132.933} C_DIS
LIN {X 0.150,Y -561.084,Z 1449.533,A 0.000,B 0.000,C 90.000,E1 131.838} C_DIS
LIN {X 0.211,Y -561.149,Z 1449.523,A 0.000,B 0.000,C 90.000,E1 130.172} C_DIS
LIN {X -0.085,Y -561.256,Z 1449.514,A 0.000,B 0.000,C 90.000,E1 128.543} C_DIS
LIN {X 0.058,Y -561.271,Z 1449.505,A 0.000,B 0.000,C 90.000,E1 126.870} C_DIS
LIN {X -0.239,Y -561.092,Z 1449.497,A 0.000,B 0.000,C 90.000,E1 125.518} C_DIS
LIN {X -0.179,Y -560.879,Z 1449.491,A 0.000,B 0.000,C 90.000,E1 124.405} C_DIS
LIN {X -0.163,Y -560.472,Z 1449.480,A 0.000,B 0.000,C 90.000,E1 122.467} C_DIS
LIN {X 0.006,Y -560.334,Z 1449.470,A 0.000,B 0.000,C 90.000,E1 120.512} C_DIS
LIN {X -0.241,Y -560.809,Z 1449.454,A 0.000,B 0.000,C 90.000,E1 117.769} C_DIS
LIN {X -0.185,Y -561.275,Z 1449.445,A 0.000,B 0.000,C 90.000,E1 116.104} C_DIS
LIN {X -0.047,Y -561.908,Z 1449.434,A 0.000,B 0.000,C 90.000,E1 114.155} C_DIS
LIN {X -0.010,Y -562.380,Z 1449.427,A 0.000,B 0.000,C 90.000,E1 112.770} C_DIS
LIN {X 0.013,Y -562.788,Z 1449.420,A 0.000,B 0.000,C 90.000,E1 111.663} C_DIS
LIN {X 0.076,Y -563.448,Z 1449.408,A 0.000,B 0.000,C 90.000,E1 109.450} C_DIS
LIN {X -0.115,Y -564.632,Z 1449.397,A 0.000,B 0.000,C 90.000,E1 107.402} C_DIS
LIN {X -0.226,Y -565.071,Z 1449.396,A 0.000,B 0.000,C 90.000,E1 107.275} C_DIS
LIN {X -0.185,Y -565.633,Z 1449.394,A 0.000,B 0.000,C 90.000,E1 106.858} C_DIS
LIN {X 0.098,Y -566.289,Z 1449.392,A 0.000,B 0.000,C 90.000,E1 106.496} C_DIS
LIN {X -0.121,Y -568.238,Z 1449.389,A 0.000,B 0.000,C 90.000,E1 105.969} C_DIS
LIN {X 0.202,Y -570.303,Z 1449.387,A 0.000,B 0.000,C 90.000,E1 105.662} C_DIS
LIN {X -0.171,Y -572.166,Z 1449.386,A 0.000,B 0.000,C 90.000,E1 105.426} C_DIS
LIN {X 0.086,Y -576.526,Z 1449.383,A 0.000,B 0.000,C 90.000,E1 104.954} C_DIS
LIN {X -0.254,Y -578.710,Z 1449.382,A 0.000,B 0.000,C 90.000,E1 104.717} C_DIS
LIN {X -0.140,Y -581.097,Z 1449.379,A 0.000,B 0.000,C 90.000,E1 104.300} C_DIS
LIN {X -0.015,Y -582.689,Z 1449.377,A 0.000,B 0.000,C 90.000,E1 103.883} C_DIS
LIN {X -0.120,Y -584.141,Z 1449.374,A 0.000,B 0.000,C 90.000,E1 103.355} C_DIS
LIN {X 0.118,Y -584.654,Z 1449.373,A 0.000,B 0.000,C 90.000,E1 103.063} C_DIS
LIN {X -0.049,Y -585.730,Z 1449.367,A 0.000,B 0.000,C 90.000,E1 102.007} C_DIS
LIN {X -0.128,Y -585.767,Z 1449.364,A 0.000,B 0.000,C 90.000,E1 101.478} C_DIS
LIN {X -0.208,Y -585.412,Z 1449.361,A 0.000,B 0.000,C 90.000,E1 100.950} C_DIS
LIN {X 0.039,Y -585.097,Z 1449.359,A 0.000,B 0.000,C 90.000,E1 100.658} C_DIS
LIN {X -0.151,Y -583.951,Z 1449.356,A 0.000,B 0.000,C 90.000,E1 100.141} C_DIS
LIN {X -0.244,Y -582.134,Z 1449.353,A 0.000,B 0.000,C 90.000,E1 99.613} C_DIS
LIN {X 0.004,Y -579.355,Z 1449.350,A 0.000,B 0.000,C 90.000,E1 98.916} C_DIS
LIN {X -0.215,Y -576.388,Z 1449.347,A 0.000,B 0.000,C 90.000,E1 98.398} C_DIS
LIN {X -0.025,Y -573.027,Z 1449.343,A 0.000,B 0.000,C 90.000,E1 97.701} C_DIS
LIN {X -0.010,Y -571.444,Z 1449.341,A 0.000,B 0.000,C 90.000,E1 97.296} C_DIS
LIN {X -0.050,Y -570.416,Z 1449.338,A 0.000,B 0.000,C 90.000,E1 96.891} C_DIS
LIN {X -0.045,Y -570.274,Z 1449.337,A 0.000,B 0.000,C 90.000,E1 96.720} C_DIS
LIN {X 0.134,Y -569.641,Z 1449.336,A 0.000,B 0.000,C 90.000,E1 96.429} C_DIS
LIN {X -0.226,Y -569.546,Z 1449.334,A 0.000,B 0.000,C 90.000,E1 96.201} C_DIS
LIN {X -0.053,Y -569.244,Z 1449.333,A 0.000,B 0.000,C 90.000,E1 95.910} C_DIS
LIN {X -0.222,Y -569.214,Z 1449.328,A 0.000,B 0.000,C 90.000,E1 95.106} C_DIS
LIN {X 0.123,Y -571.206,Z 1449.312,A 0.000,B 0.000,C 90.000,E1 92.064} C_DIS
LIN {X -0.191,Y -572.617,Z 1449.302,A 0.000,B 0.000,C 90.000,E1 90.458} C_DIS
LIN {X 0.083,Y -574.003,Z 1449.293,A 0.000,B 0.000,C 90.000,E1 88.797} C_DIS
LIN {X 0.251,Y -575.186,Z 1449.286,A 0.000,B 0.000,C 90.000,E1 87.421} C_DIS
LIN {X 0.051,Y -576.666,Z 1449.277,A 0.000,B 0.000,C 90.000,E1 85.812} C_DIS
LIN {X 0.227,Y -578.651,Z 1449.265,A 0.000,B 0.000,C 90.000,E1 83.628} C_DIS
LIN {X 0.219,Y -580.118,Z 1449.256,A 0.000,B 0.000,C 90.000,E1 82.008} C_DIS
LIN {X 0.016,Y -581.455,Z 1449.248,A 0.000,B 0.000,C 90.000,E1 80.679} C_DIS
LIN {X 0.158,Y -583.049,Z 1449.239,A 0.000,B 0.000,C 90.000,E1 79.050} C_DIS
LIN {X -0.123,Y -584.657,Z 1449.230,A 0.000,B 0.000,C 90.000,E1 77.465} C_DIS
LIN {X 0.193,Y -585.950,Z 1449.221,A 0.000,B 0.000,C 90.000,E1 75.825} C_DIS
LIN {X -0.143,Y -586.915,Z 1449.214,A 0.000,B 0.000,C 90.000,E1 74.519} C_DIS
LIN {X 0.035,Y -588.154,Z 1449.202,A 0.000,B 0.000,C 90.000,E1 72.362} C_DIS
LIN {X -0.229,Y -588.986,Z 1449.193,A 0.000,B 0.000,C 90.000,E1 70.786} C_DIS
LIN {X 0.074,Y -589.769,Z 1449.184,A 0.000,B 0.000,C 90.000,E1 69.156} C_DIS
LIN {X 0.259,Y -590.701,Z 1449.175,A 0.000,B 0.000,C 90.000,E1 67.539} C_DIS
LIN {X 0.037,Y -591.467,Z 1449.168,A 0.000,B 0.000,C 90.000,E1 66.230} C_DIS
LIN {X 0.270,Y -591.869,Z 1449.164,A 0.000,B 0.000,C 90.000,E1 65.409} C_DIS
LIN {X -0.140,Y -593.274,Z 1449.153,A 0.000,B 0.000,C 90.000,E1 63.589} C_DIS
LIN {X -0.005,Y -594.586,Z 1449.143,A 0.000,B 0.000,C 90.000,E1 61.719} C_DIS
LIN {X -0.163,Y -596.387,Z 1449.131,A 0.000,B 0.000,C 90.000,E1 59.616} C_DIS
LIN {X 0.115,Y -598.017,Z 1449.121,A 0.000,B 0.000,C 90.000,E1 57.740} C_DIS
LIN {X 0.113,Y -599.190,Z 1449.114,A 0.000,B 0.000,C 90.000,E1 56.421} C_DIS
LIN {X 0.039,Y -600.638,Z 1449.105,A 0.000,B 0.000,C 90.000,E1 54.848} C_DIS
LIN {X -0.054,Y -601.633,Z 1449.098,A 0.000,B 0.000,C 90.000,E1 53.543} C_DIS
LIN {X -0.231,Y -602.742,Z 1449.089,A 0.000,B 0.000,C 90.000,E1 51.984} C_DIS
LIN {X 0.097,Y -603.554,Z 1449.081,A 0.000,B 0.000,C 90.000,E1 50.642} C_DIS
LIN {X -0.200,Y -604.089,Z 1449.076,A 0.000,B 0.000,C 90.000,E1 49.622} C_DIS
LIN {X -0.107,Y -604.286,Z 1449.070,A 0.000,B 0.000,C 90.000,E1 48.566} C_DIS
LIN {X -0.005,Y -604.597,Z 1449.061,A 0.000,B 0.000,C 90.000,E1 46.986} C_DIS
LIN {X -0.353,Y -604.766,Z 1449.055,A 0.000,B 0.000,C 90.000,E1 45.972} C_DIS
LIN {X -0.280,Y -604.608,Z 1449.049,A 0.000,B 0.000,C 90.000,E1 44.919} C_DIS
LIN {X -0.013,Y -604.310,Z 1449.045,A 0.000,B 0.000,C 90.000,E1 44.109} C_DIS
LIN {X 0.249,Y -603.854,Z 1449.041,A 0.000,B 0.000,C 90.000,E1 43.299} C_DIS
LIN {X 0.131,Y -602.887,Z 1449.033,A 0.000,B 0.000,C 90.000,E1 42.000} C_DIS
LIN {X -0.243,Y -601.949,Z 1449.028,A 0.000,B 0.000,C 90.000,E1 40.987} C_DIS
LIN {X -0.180,Y -600.812,Z 1449.022,A 0.000,B 0.000,C 90.000,E1 39.930} C_DIS
LIN {X 0.329,Y -599.446,Z 1449.016,A 0.000,B 0.000,C 90.000,E1 38.830} C_DIS
LIN {X 0.217,Y -597.559,Z 1449.009,A 0.000,B 0.000,C 90.000,E1 37.523} C_DIS
LIN {X 0.086,Y -596.323,Z 1449.004,A 0.000,B 0.000,C 90.000,E1 36.744} C_DIS
LIN {X 0.069,Y -595.284,Z 1449.001,A 0.000,B 0.000,C 90.000,E1 36.217} C_DIS
LIN {X 0.132,Y -593.050,Z 1448.995,A 0.000,B 0.000,C 90.000,E1 35.152} C_DIS
LIN {X 0.029,Y -589.804,Z 1448.988,A 0.000,B 0.000,C 90.000,E1 33.833} C_DIS
LIN {X -0.022,Y -587.563,Z 1448.984,A 0.000,B 0.000,C 90.000,E1 33.038} C_DIS
LIN {X 0.098,Y -584.358,Z 1448.978,A 0.000,B 0.000,C 90.000,E1 31.957} C_DIS
LIN {X 0.143,Y -582.551,Z 1448.975,A 0.000,B 0.000,C 90.000,E1 31.416} C_DIS
LIN {X 0.172,Y -580.550,Z 1448.972,A 0.000,B 0.000,C 90.000,E1 30.875} C_DIS
LIN {X 0.186,Y -578.276,Z 1448.969,A 0.000,B 0.000,C 90.000,E1 30.335} C_DIS
LIN {X -0.129,Y -573.211,Z 1448.963,A 0.000,B 0.000,C 90.000,E1 29.283} C_DIS
LIN {X -0.260,Y -569.668,Z 1448.959,A 0.000,B 0.000,C 90.000,E1 28.615} C_DIS
LIN {X -0.015,Y -565.134,Z 1448.954,A 0.000,B 0.000,C 90.000,E1 27.769} C_DIS
LIN {X -0.079,Y -560.311,Z 1448.950,A 0.000,B 0.000,C 90.000,E1 26.950} C_DIS
LIN {X 0.166,Y -555.976,Z 1448.946,A 0.000,B 0.000,C 90.000,E1 26.232} C_DIS
LIN {X 0.123,Y -551.291,Z 1448.942,A 0.000,B 0.000,C 90.000,E1 25.540} C_DIS
LIN {X -0.217,Y -548.319,Z 1448.940,A 0.000,B 0.000,C 90.000,E1 25.155} C_DIS
LIN {X -0.198,Y -544.068,Z 1448.937,A 0.000,B 0.000,C 90.000,E1 24.591} C_DIS
LIN {X -0.121,Y -538.454,Z 1448.933,A 0.000,B 0.000,C 90.000,E1 23.875} C_DIS
LIN {X -0.181,Y -531.282,Z 1448.928,A 0.000,B 0.000,C 90.000,E1 23.025} C_DIS
LIN {X -0.085,Y -523.707,Z 1448.923,A 0.000,B 0.000,C 90.000,E1 22.153} C_DIS
LIN {X 0.156,Y -517.209,Z 1448.919,A 0.000,B 0.000,C 90.000,E1 21.408} C_DIS
LIN {X 0.050,Y -507.925,Z 1448.914,A 0.000,B 0.000,C 90.000,E1 20.429} C_DIS
LIN {X -0.040,Y -498.706,Z 1448.908,A 0.000,B 0.000,C 90.000,E1 19.504} C_DIS
LIN {X 0.052,Y -484.246,Z 1448.900,A 0.000,B 0.000,C 90.000,E1 18.000} C_DIS
LIN {X -0.167,Y -478.709,Z 1448.897,A 0.000,B 0.000,C 90.000,E1 17.457} C_DIS
LIN {X 0.187,Y -472.726,Z 1448.894,A 0.000,B 0.000,C 90.000,E1 16.858} C_DIS
LIN {X -0.056,Y -467.848,Z 1448.892,A 0.000,B 0.000,C 90.000,E1 16.496} C_DIS
LIN {X -0.054,Y -464.302,Z 1448.890,A 0.000,B 0.000,C 90.000,E1 16.260} C_DIS
LIN {X 0.122,Y -462.369,Z 1448.890,A 0.000,B 0.000,C 90.000,E1 16.134} C_DIS
LIN {X 0.062,Y -458.999,Z 1448.889,A 0.000,B 0.000,C 90.000,E1 16.024} C_DIS
LIN {X -0.016,Y -458.192,Z 1448.889,A 0.000,B 0.000,C 90.000,E1 16.024} C_DIS
LIN {X -0.034,Y -371.712,Z 1448.889,A 0.000,B 0.000,C 90.000,E1 16.024} C_DIS
LIN {X 0.050,Y -366.723,Z 1448.858,A 0.000,B 0.000,C 90.000,E1 10.366} C_DIS
LIN {X -0.093,Y -366.527,Z 1448.856,A 0.000,B 0.000,C 90.000,E1 10.018} C_DIS
LIN {X 0.050,Y -365.032,Z 1448.847,A 0.000,B 0.000,C 90.000,E1 8.511} C_DIS
LIN {X 0.146,Y -361.083,Z 1448.810,A 0.000,B 0.000,C 90.000,E1 1.776} C_DIS
LIN {X 0.086,Y -360.905,Z 1448.802,A 0.000,B 0.000,C 90.000,E1 0.286} C_DIS
LIN {X -0.053,Y -359.426,Z 1448.770,A 0.000,B 0.000,C 90.000,E1 354.546} C_DIS
LIN {X 0.070,Y -358.890,Z 1448.759,A 0.000,B 0.000,C 90.000,E1 352.648} C_DIS
LIN {X -0.020,Y -359.563,Z 1448.726,A 0.000,B 0.000,C 90.000,E1 346.645} C_DIS
LIN {X 0.001,Y -361.801,Z 1448.684,A 0.000,B 0.000,C 90.000,E1 339.135} C_DIS
LIN {X -0.154,Y -362.053,Z 1448.680,A 0.000,B 0.000,C 90.000,E1 338.411} C_DIS
LIN {X 0.189,Y -365.980,Z 1448.643,A 0.000,B 0.000,C 90.000,E1 331.641} C_DIS
LIN {X 0.029,Y -366.387,Z 1448.639,A 0.000,B 0.000,C 90.000,E1 330.923} C_DIS
LIN {X -0.031,Y -371.355,Z 1448.604,A 0.000,B 0.000,C 90.000,E1 324.642} C_DIS
LIN {X -0.043,Y -371.766,Z 1448.602,A 0.000,B 0.000,C 90.000,E1 324.276} C_DIS
LIN {X 0.013,Y -377.358,Z 1448.567,A 0.000,B 0.000,C 90.000,E1 318.038} C_DIS
LIN {X 0.012,Y -378.235,Z 1448.563,A 0.000,B 0.000,C 90.000,E1 317.310} C_DIS
LIN {X 0.002,Y -383.940,Z 1448.531,A 0.000,B 0.000,C 90.000,E1 311.515} C_DIS
LIN {X 0.088,Y -384.893,Z 1448.527,A 0.000,B 0.000,C 90.000,E1 310.782} C_DIS
LIN {X 0.262,Y -390.610,Z 1448.495,A 0.000,B 0.000,C 90.000,E1 305.025} C_DIS
LIN {X 0.106,Y -391.104,Z 1448.493,A 0.000,B 0.000,C 90.000,E1 304.692} C_DIS
LIN {X 0.022,Y -391.648,Z 1448.489,A 0.000,B 0.000,C 90.000,E1 303.992} C_DIS
LIN {X -0.080,Y -396.825,Z 1448.459,A 0.000,B 0.000,C 90.000,E1 298.693} C_DIS
LIN {X -0.210,Y -397.120,Z 1448.457,A 0.000,B 0.000,C 90.000,E1 298.359} C_DIS
LIN {X -0.055,Y -401.597,Z 1448.426,A 0.000,B 0.000,C 90.000,E1 292.717} C_DIS
LIN {X 0.222,Y -404.659,Z 1448.395,A 0.000,B 0.000,C 90.000,E1 287.094} C_DIS
LIN {X -0.079,Y -404.735,Z 1448.391,A 0.000,B 0.000,C 90.000,E1 286.441} C_DIS
LIN {X 0.214,Y -406.099,Z 1448.364,A 0.000,B 0.000,C 90.000,E1 281.535} C_DIS
LIN {X -0.176,Y -406.094,Z 1448.362,A 0.000,B 0.000,C 90.000,E1 281.243} C_DIS
LIN {X -0.097,Y -405.680,Z 1448.333,A 0.000,B 0.000,C 90.000,E1 276.024} C_DIS
LIN {X -0.165,Y -405.058,Z 1448.328,A 0.000,B 0.000,C 90.000,E1 274.992} C_DIS
LIN {X -0.060,Y -403.497,Z 1448.304,A 0.000,B 0.000,C 90.000,E1 270.802} C_DIS
LIN {X -0.092,Y -403.288,Z 1448.302,A 0.000,B 0.000,C 90.000,E1 270.458} C_DIS
LIN {X 0.091,Y -398.931,Z 1448.271,A 0.000,B 0.000,C 90.000,E1 264.837} C_DIS
LIN {X -0.040,Y -393.108,Z 1448.242,A 0.000,B 0.000,C 90.000,E1 259.567} C_DIS
LIN {X -0.079,Y -392.835,Z 1448.240,A 0.000,B 0.000,C 90.000,E1 259.218} C_DIS
LIN {X 0.034,Y -385.993,Z 1448.212,A 0.000,B 0.000,C 90.000,E1 254.212} C_DIS
LIN {X -0.026,Y -385.267,Z 1448.208,A 0.000,B 0.000,C 90.000,E1 253.504} C_DIS
LIN {X -0.004,Y -384.768,Z 1448.206,A 0.000,B 0.000,C 90.000,E1 253.142} C_DIS
LIN {X 0.221,Y -377.973,Z 1448.182,A 0.000,B 0.000,C 90.000,E1 248.773} C_DIS
LIN {X -0.044,Y -376.233,Z 1448.174,A 0.000,B 0.000,C 90.000,E1 247.358} C_DIS
LIN {X 0.057,Y -374.944,Z 1448.170,A 0.000,B 0.000,C 90.000,E1 246.613} C_DIS
LIN {X -0.208,Y -368.417,Z 1448.148,A 0.000,B 0.000,C 90.000,E1 242.615} C_DIS
LIN {X 0.097,Y -366.047,Z 1448.137,A 0.000,B 0.000,C 90.000,E1 240.717} C_DIS
LIN {X 0.004,Y -359.196,Z 1448.115,A 0.000,B 0.000,C 90.000,E1 236.628} C_DIS
LIN {X 0.021,Y -355.842,Z 1448.100,A 0.000,B 0.000,C 90.000,E1 233.989} C_DIS
LIN {X -0.173,Y -348.793,Z 1448.075,A 0.000,B 0.000,C 90.000,E1 229.461} C_DIS
LIN {X -0.097,Y -346.185,Z 1448.062,A 0.000,B 0.000,C 90.000,E1 227.148} C_DIS
LIN {X -0.088,Y -345.065,Z 1448.058,A 0.000,B 0.000,C 90.000,E1 226.377} C_DIS
LIN {X 0.094,Y -338.586,Z 1448.030,A 0.000,B 0.000,C 90.000,E1 221.310} C_DIS
LIN {X 0.094,Y -336.840,Z 1448.019,A 0.000,B 0.000,C 90.000,E1 219.358} C_DIS
LIN {X 0.014,Y -330.861,Z 1447.988,A 0.000,B 0.000,C 90.000,E1 213.865} C_DIS
LIN {X 0.149,Y -329.296,Z 1447.975,A 0.000,B 0.000,C 90.000,E1 211.465} C_DIS
LIN {X -0.154,Y -324.669,Z 1447.942,A 0.000,B 0.000,C 90.000,E1 205.540} C_DIS
LIN {X 0.174,Y -323.837,Z 1447.928,A 0.000,B 0.000,C 90.000,E1 203.078} C_DIS
LIN {X -0.017,Y -321.124,Z 1447.881,A 0.000,B 0.000,C 90.000,E1 194.662} C_DIS
LIN {X 0.138,Y -320.932,Z 1447.877,A 0.000,B 0.000,C 90.000,E1 193.828} C_DIS
LIN {X -0.076,Y -321.562,Z 1447.832,A 0.000,B 0.000,C 90.000,E1 185.796} C_DIS
LIN {X -0.143,Y -324.415,Z 1447.790,A 0.000,B 0.000,C 90.000,E1 178.165} C_DIS
LIN {X -0.141,Y -325.376,Z 1447.783,A 0.000,B 0.000,C 90.000,E1 176.963} C_DIS
LIN {X -0.100,Y -329.112,Z 1447.750,A 0.000,B 0.000,C 90.000,E1 170.971} C_DIS
LIN {X 0.061,Y -334.260,Z 1447.726,A 0.000,B 0.000,C 90.000,E1 166.589} C_DIS
LIN {X 0.067,Y -335.488,Z 1447.719,A 0.000,B 0.000,C 90.000,E1 165.408} C_DIS
LIN {X 0.191,Y -339.266,Z 1447.702,A 0.000,B 0.000,C 90.000,E1 162.236} C_DIS
LIN {X 0.189,Y -402.592,Z 1447.702,A 0.000,B 0.000,C 90.000,E1 162.236} C_DIS
LIN {X 0.010,Y -406.057,Z 1447.701,A 0.000,B 0.000,C 90.000,E1 162.181} C_DIS
LIN {X 0.036,Y -410.245,Z 1447.700,A 0.000,B 0.000,C 90.000,E1 162.000} C_DIS
LIN {X 0.054,Y -415.344,Z 1447.698,A 0.000,B 0.000,C 90.000,E1 161.710} C_DIS
LIN {X 0.166,Y -421.507,Z 1447.696,A 0.000,B 0.000,C 90.000,E1 161.275} C_DIS
LIN {X 0.237,Y -427.697,Z 1447.693,A 0.000,B 0.000,C 90.000,E1 160.786} C_DIS
LIN {X -0.058,Y -441.527,Z 1447.687,A 0.000,B 0.000,C 90.000,E1 159.645} C_DIS
LIN {X 0.085,Y -455.285,Z 1447.680,A 0.000,B 0.000,C 90.000,E1 158.465} C_DIS
LIN {X -0.081,Y -465.958,Z 1447.676,A 0.000,B 0.000,C 90.000,E1 157.592} C_DIS
LIN {X 0.115,Y -477.632,Z 1447.670,A 0.000,B 0.000,C 90.000,E1 156.561} C_DIS
LIN {X 0.036,Y -484.916,Z 1447.666,A 0.000,B 0.000,C 90.000,E1 155.921} C_DIS
LIN {X 0.194,Y -493.575,Z 1447.662,A 0.000,B 0.000,C 90.000,E1 155.101} C_DIS
LIN {X -0.154,Y -500.428,Z 1447.658,A 0.000,B 0.000,C 90.000,E1 154.460} C_DIS
LIN {X -0.157,Y -505.756,Z 1447.655,A 0.000,B 0.000,C 90.000,E1 153.896} C_DIS
LIN {X -0.097,Y -509.612,Z 1447.653,A 0.000,B 0.000,C 90.000,E1 153.461} C_DIS
LIN {X -0.131,Y -514.464,Z 1447.649,A 0.000,B 0.000,C 90.000,E1 152.871} C_DIS
LIN {X 0.045,Y -517.893,Z 1447.647,A 0.000,B 0.000,C 90.000,E1 152.410} C_DIS
LIN {X -0.167,Y -521.892,Z 1447.644,A 0.000,B 0.000,C 90.000,E1 151.847} C_DIS
LIN {X -0.014,Y -526.284,Z 1447.640,A 0.000,B 0.000,C 90.000,E1 151.101} C_DIS
LIN {X -0.175,Y -529.472,Z 1447.636,A 0.000,B 0.000,C 90.000,E1 150.539} C_DIS
LIN {X 0.060,Y -532.885,Z 1447.632,A 0.000,B 0.000,C 90.000,E1 149.793} C_DIS
LIN {X 0.349,Y -534.797,Z 1447.630,A 0.000,B 0.000,C 90.000,E1 149.331} C_DIS
LIN {X -0.242,Y -538.107,Z 1447.625,A 0.000,B 0.000,C 90.000,E1 148.535} C_DIS
LIN {X -0.063,Y -541.048,Z 1447.620,A 0.000,B 0.000,C 90.000,E1 147.661} C_DIS
LIN {X -0.034,Y -542.796,Z 1447.617,A 0.000,B 0.000,C 90.000,E1 147.089} C_DIS
LIN {X -0.074,Y -545.903,Z 1447.611,A 0.000,B 0.000,C 90.000,E1 145.960} C_DIS
LIN {X 0.042,Y -547.980,Z 1447.606,A 0.000,B 0.000,C 90.000,E1 145.102} C_DIS
LIN {X -0.182,Y -549.280,Z 1447.603,A 0.000,B 0.000,C 90.000,E1 144.562} C_DIS
LIN {X 0.033,Y -551.411,Z 1447.597,A 0.000,B 0.000,C 90.000,E1 143.417} C_DIS
LIN {X 0.282,Y -553.183,Z 1447.591,A 0.000,B 0.000,C 90.000,E1 142.271} C_DIS
LIN {X -0.020,Y -554.013,Z 1447.588,A 0.000,B 0.000,C 90.000,E1 141.743} C_DIS
LIN {X -0.099,Y -555.612,Z 1447.580,A 0.000,B 0.000,C 90.000,E1 140.356} C_DIS
LIN {X 0.128,Y -556.693,Z 1447.574,A 0.000,B 0.000,C 90.000,E1 139.218} C_DIS
LIN {X 0.031,Y -557.899,Z 1447.566,A 0.000,B 0.000,C 90.000,E1 137.838} C_DIS
LIN {X -0.052,Y -558.945,Z 1447.558,A 0.000,B 0.000,C 90.000,E1 136.458} C_DIS
LIN {X 0.193,Y -559.700,Z 1447.552,A 0.000,B 0.000,C 90.000,E1 135.324} C_DIS
LIN {X -0.342,Y -560.281,Z 1447.546,A 0.000,B 0.000,C 90.000,E1 134.271} C_DIS
LIN {X -0.081,Y -560.740,Z 1447.540,A 0.000,B 0.000,C 90.000,E1 133.137} C_DIS
LIN {X 0.213,Y -561.081,Z 1447.533,A 0.000,B 0.000,C 90.000,E1 132.000} C_DIS
LIN {X -0.030,Y -561.141,Z 1447.530,A 0.000,B 0.000,C 90.000,E1 131.472} C_DIS
LIN {X -0.206,Y -561.230,Z 1447.518,A 0.000,B 0.000,C 90.000,E1 129.277} C_DIS
LIN {X -0.160,Y -561.244,Z 1447.510,A 0.000,B 0.000,C 90.000,E1 127.890} C_DIS
LIN {X -0.215,Y -561.250,Z 1447.504,A 0.000,B 0.000,C 90.000,E1 126.790} C_DIS
LIN {X 0.038,Y -561.030,Z 1447.495,A 0.000,B 0.000,C 90.000,E1 125.105} C_DIS
LIN {X 0.192,Y -560.717,Z 1447.487,A 0.000,B 0.000,C 90.000,E1 123.706} C_DIS
LIN {X 0.026,Y -560.452,Z 1447.480,A 0.000,B 0.000,C 90.000,E1 122.339} C_DIS
LIN {X 0.120,Y -560.351,Z 1447.470,A 0.000,B 0.000,C 90.000,E1 120.669} C_DIS
LIN {X -0.046,Y -560.846,Z 1447.454,A 0.000,B 0.000,C 90.000,E1 117.641} C_DIS
LIN {X 0.011,Y -561.338,Z 1447.444,A 0.000,B 0.000,C 90.000,E1 115.976} C_DIS
LIN {X 0.151,Y -561.957,Z 1447.434,A 0.000,B 0.000,C 90.000,E1 114.027} C_DIS
LIN {X -0.015,Y -562.531,Z 1447.424,A 0.000,B 0.000,C 90.000,E1 112.386} C_DIS
LIN {X 0.209,Y -562.834,Z 1447.420,A 0.000,B 0.000,C 90.000,E1 111.535} C_DIS
LIN {X -0.205,Y -564.083,Z 1447.403,A 0.000,B 0.000,C 90.000,E1 108.544} C_DIS
LIN {X 0.113,Y -564.475,Z 1447.401,A 0.000,B 0.000,C 90.000,E1 108.236} C_DIS
LIN {X -0.240,Y -565.071,Z 1447.398,A 0.000,B 0.000,C 90.000,E1 107.583} C_DIS
LIN {X -0.031,Y -566.341,Z 1447.395,A 0.000,B 0.000,C 90.000,E1 107.149} C_DIS
LIN {X -0.211,Y -566.449,Z 1447.395,A 0.000,B 0.000,C 90.000,E1 107.094} C_DIS
LIN {X -0.253,Y -566.456,Z 1447.395,A 0.000,B 0.000,C 90.000,E1 107.094} C_DIS
LIN {X -0.257,Y -568.942,Z 1447.392,A 0.000,B 0.000,C 90.000,E1 106.622} C_DIS
LIN {X 0.146,Y -574.648,Z 1447.389,A 0.000,B 0.000,C 90.000,E1 106.024} C_DIS
LIN {X 0.019,Y -579.932,Z 1447.386,A 0.000,B 0.000,C 90.000,E1 105.552} C_DIS
LIN {X 0.031,Y -582.565,Z 1447.385,A 0.000,B 0.000,C 90.000,E1 105.300} C_DIS
LIN {X -0.121,Y -583.591,Z 1447.384,A 0.000,B 0.000,C 90.000,E1 105.190} C_DIS
LIN {X 0.262,Y -587.340,Z 1447.381,A 0.000,B 0.000,C 90.000,E1 104.481} C_DIS
LIN {X 0.173,Y -587.929,Z 1447.380,A 0.000,B 0.000,C 90.000,E1 104.356} C_DIS
LIN {X 0.106,Y -589.370,Z 1447.377,A 0.000,B 0.000,C 90.000,E1 103.828} C_DIS
LIN {X -0.262,Y -590.741,Z 1447.372,A 0.000,B 0.000,C 90.000,E1 103.063} C_DIS
LIN {X -0.307,Y -591.346,Z 1447.370,A 0.000,B 0.000,C 90.000,E1 102.535} C_DIS
LIN {X -0.076,Y -591.547,Z 1447.365,A 0.000,B 0.000,C 90.000,E1 101.715} C_DIS
LIN {X -0.114,Y -591.354,Z 1447.362,A 0.000,B 0.000,C 90.000,E1 101.186} C_DIS
LIN {X -0.156,Y -590.812,Z 1447.359,A 0.000,B 0.000,C 90.000,E1 100.658} C_DIS
LIN {X -0.307,Y -589.466,Z 1447.356,A 0.000,B 0.000,C 90.000,E1 100.141} C_DIS
LIN {X 0.219,Y -587.798,Z 1447.353,A 0.000,B 0.000,C 90.000,E1 99.557} C_DIS
LIN {X 0.148,Y -585.724,Z 1447.350,A 0.000,B 0.000,C 90.000,E1 99.029} C_DIS
LIN {X -0.272,Y -584.550,Z 1447.349,A 0.000,B 0.000,C 90.000,E1 98.803} C_DIS
LIN {X 0.207,Y -581.530,Z 1447.346,A 0.000,B 0.000,C 90.000,E1 98.219} C_DIS
LIN {X -0.004,Y -575.373,Z 1447.341,A 0.000,B 0.000,C 90.000,E1 97.296} C_DIS
LIN {X -0.089,Y -572.931,Z 1447.338,A 0.000,B 0.000,C 90.000,E1 96.777} C_DIS
LIN {X -0.122,Y -570.858,Z 1447.335,A 0.000,B 0.000,C 90.000,E1 96.372} C_DIS
LIN {X 0.061,Y -570.541,Z 1447.335,A 0.000,B 0.000,C 90.000,E1 96.258} C_DIS
LIN {X 0.184,Y -569.818,Z 1447.332,A 0.000,B 0.000,C 90.000,E1 95.739} C_DIS
LIN {X 0.086,Y -569.773,Z 1447.331,A 0.000,B 0.000,C 90.000,E1 95.568} C_DIS
LIN {X 0.257,Y -569.509,Z 1447.329,A 0.000,B 0.000,C 90.000,E1 95.277} C_DIS
LIN {X -0.027,Y -569.490,Z 1447.326,A 0.000,B 0.000,C 90.000,E1 94.759} C_DIS
LIN {X -0.127,Y -571.725,Z 1447.308,A 0.000,B 0.000,C 90.000,E1 91.489} C_DIS
LIN {X 0.268,Y -573.401,Z 1447.298,A 0.000,B 0.000,C 90.000,E1 89.542} C_DIS
LIN {X 0.145,Y -575.050,Z 1447.287,A 0.000,B 0.000,C 90.000,E1 87.650} C_DIS
LIN {X 0.091,Y -576.772,Z 1447.276,A 0.000,B 0.000,C 90.000,E1 85.755} C_DIS
LIN {X 0.269,Y -578.766,Z 1447.265,A 0.000,B 0.000,C 90.000,E1 83.571} C_DIS
LIN {X 0.042,Y -580.012,Z 1447.257,A 0.000,B 0.000,C 90.000,E1 82.243} C_DIS
LIN {X -0.075,Y -581.350,Z 1447.250,A 0.000,B 0.000,C 90.000,E1 80.905} C_DIS
LIN {X 0.201,Y -583.215,Z 1447.239,A 0.000,B 0.000,C 90.000,E1 78.993} C_DIS
LIN {X -0.080,Y -584.815,Z 1447.230,A 0.000,B 0.000,C 90.000,E1 77.409} C_DIS
LIN {X -0.188,Y -586.092,Z 1447.221,A 0.000,B 0.000,C 90.000,E1 75.811} C_DIS
LIN {X 0.056,Y -587.069,Z 1447.214,A 0.000,B 0.000,C 90.000,E1 74.448} C_DIS
LIN {X 0.074,Y -588.314,Z 1447.202,A 0.000,B 0.000,C 90.000,E1 72.308} C_DIS
LIN {X 0.236,Y -589.273,Z 1447.191,A 0.000,B 0.000,C 90.000,E1 70.423} C_DIS
LIN {X 0.305,Y -590.402,Z 1447.180,A 0.000,B 0.000,C 90.000,E1 68.284} C_DIS
LIN {X -0.263,Y -591.330,Z 1447.171,A 0.000,B 0.000,C 90.000,E1 66.741} C_DIS
LIN {X -0.037,Y -591.704,Z 1447.166,A 0.000,B 0.000,C 90.000,E1 65.921} C_DIS
LIN {X 0.147,Y -593.453,Z 1447.153,A 0.000,B 0.000,C 90.000,E1 63.512} C_DIS
LIN {X -0.136,Y -594.588,Z 1447.144,A 0.000,B 0.000,C 90.000,E1 61.948} C_DIS
LIN {X 0.152,Y -596.570,Z 1447.131,A 0.000,B 0.000,C 90.000,E1 59.537} C_DIS
LIN {X -0.063,Y -598.216,Z 1447.121,A 0.000,B 0.000,C 90.000,E1 57.709} C_DIS
LIN {X -0.145,Y -599.619,Z 1447.112,A 0.000,B 0.000,C 90.000,E1 56.135} C_DIS
LIN {X -0.108,Y -600.829,Z 1447.104,A 0.000,B 0.000,C 90.000,E1 54.815} C_DIS
LIN {X -0.059,Y -601.817,Z 1447.097,A 0.000,B 0.000,C 90.000,E1 53.497} C_DIS
LIN {X 0.129,Y -602.943,Z 1447.089,A 0.000,B 0.000,C 90.000,E1 51.904} C_DIS
LIN {X 0.081,Y -603.740,Z 1447.081,A 0.000,B 0.000,C 90.000,E1 50.598} C_DIS
LIN {X 0.170,Y -604.263,Z 1447.075,A 0.000,B 0.000,C 90.000,E1 49.542} C_DIS
LIN {X -0.187,Y -604.477,Z 1447.070,A 0.000,B 0.000,C 90.000,E1 48.528} C_DIS
LIN {X -0.237,Y -604.819,Z 1447.059,A 0.000,B 0.000,C 90.000,E1 46.701} C_DIS
LIN {X 0.028,Y -604.925,Z 1447.055,A 0.000,B 0.000,C 90.000,E1 45.891} C_DIS
LIN {X 0.105,Y -604.773,Z 1447.049,A 0.000,B 0.000,C 90.000,E1 44.838} C_DIS
LIN {X 0.374,Y -604.472,Z 1447.045,A 0.000,B 0.000,C 90.000,E1 44.028} C_DIS
LIN {X -0.219,Y -604.021,Z 1447.041,A 0.000,B 0.000,C 90.000,E1 43.299} C_DIS
LIN {X 0.070,Y -603.056,Z 1447.033,A 0.000,B 0.000,C 90.000,E1 41.962} C_DIS
LIN {X 0.354,Y -602.392,Z 1447.029,A 0.000,B 0.000,C 90.000,E1 41.148} C_DIS
LIN {X -0.035,Y -601.303,Z 1447.023,A 0.000,B 0.000,C 90.000,E1 40.135} C_DIS
LIN {X 0.099,Y -600.009,Z 1447.017,A 0.000,B 0.000,C 90.000,E1 39.072} C_DIS
LIN {X 0.369,Y -598.178,Z 1447.010,A 0.000,B 0.000,C 90.000,E1 37.729} C_DIS
LIN {X -0.003,Y -596.513,Z 1447.004,A 0.000,B 0.000,C 90.000,E1 36.710} C_DIS
LIN {X -0.147,Y -594.930,Z 1447.000,A 0.000,B 0.000,C 90.000,E1 35.931} C_DIS
LIN {X 0.178,Y -593.231,Z 1446.995,A 0.000,B 0.000,C 90.000,E1 35.105} C_DIS
LIN {X 0.086,Y -589.987,Z 1446.988,A 0.000,B 0.000,C 90.000,E1 33.785} C_DIS
LIN {X -0.131,Y -587.766,Z 1446.983,A 0.000,B 0.000,C 90.000,E1 33.007} C_DIS
LIN {X -0.198,Y -585.401,Z 1446.979,A 0.000,B 0.000,C 90.000,E1 32.212} C_DIS
LIN {X 0.024,Y -582.724,Z 1446.974,A 0.000,B 0.000,C 90.000,E1 31.386} C_DIS
LIN {X 0.050,Y -580.715,Z 1446.971,A 0.000,B 0.000,C 90.000,E1 30.846} C_DIS
LIN {X -0.303,Y -577.854,Z 1446.968,A 0.000,B 0.000,C 90.000,E1 30.207} C_DIS
LIN {X 0.159,Y -572.742,Z 1446.962,A 0.000,B 0.000,C 90.000,E1 29.077} C_DIS
LIN {X -0.152,Y -567.654,Z 1446.956,A 0.000,B 0.000,C 90.000,E1 28.153} C_DIS
LIN {X -0.028,Y -562.144,Z 1446.951,A 0.000,B 0.000,C 90.000,E1 27.180} C_DIS
LIN {X -0.021,Y -557.934,Z 1446.947,A 0.000,B 0.000,C 90.000,E1 26.488} C_DIS
LIN {X -0.045,Y -553.456,Z 1446.943,A 0.000,B 0.000,C 90.000,E1 25.796} C_DIS
LIN {X 0.128,Y -548.557,Z 1446.939,A 0.000,B 0.000,C 90.000,E1 25.079} C_DIS
LIN {X 0.019,Y -543.246,Z 1446.936,A 0.000,B 0.000,C 90.000,E1 24.387} C_DIS
LIN {X -0.066,Y -537.624,Z 1446.932,A 0.000,B 0.000,C 90.000,E1 23.695} C_DIS
LIN {X 0.115,Y -530.408,Z 1446.927,A 0.000,B 0.000,C 90.000,E1 22.823} C_DIS
LIN {X 0.066,Y -522.846,Z 1446.922,A 0.000,B 0.000,C 90.000,E1 21.972} C_DIS
LIN {X -0.027,Y -517.618,Z 1446.919,A 0.000,B 0.000,C 90.000,E1 21.408} C_DIS
LIN {X -0.106,Y -508.355,Z 1446.913,A 0.000,B 0.000,C 90.000,E1 20.429} C_DIS
LIN {X 0.229,Y -499.174,Z 1446.908,A 0.000,B 0.000,C 90.000,E1 19.450} C_DIS
LIN {X -0.075,Y -483.501,Z 1446.899,A 0.000,B 0.000,C 90.000,E1 17.873} C_DIS
LIN {X -0.057,Y -473.927,Z 1446.894,A 0.000,B 0.000,C 90.000,E1 16.858} C_DIS
LIN {X -0.183,Y -469.492,Z 1446.891,A 0.000,B 0.000,C 90.000,E1 16.441} C_DIS
LIN {X -0.085,Y -464.842,Z 1446.889,A 0.000,B 0.000,C 90.000,E1 16.024} C_DIS
LIN {X -0.219,Y -461.478,Z 1446.888,A 0.000,B 0.000,C 90.000,E1 15.788} C_DIS
LIN {X -0.164,Y -457.759,Z 1446.886,A 0.000,B 0.000,C 90.000,E1 15.552} C_DIS
LIN {X -0.024,Y -455.339,Z 1446.886,A 0.000,B 0.000,C 90.000,E1 15.426} C_DIS
LIN {X 0.164,Y -454.329,Z 1446.885,A 0.000,B 0.000,C 90.000,E1 15.371} C_DIS
LIN {X -0.037,Y -452.763,Z 1446.885,A 0.000,B 0.000,C 90.000,E1 15.371} C_DIS
LIN {X -0.064,Y -370.932,Z 1446.885,A 0.000,B 0.000,C 90.000,E1 15.371} C_DIS
LIN {X 0.132,Y -366.574,Z 1446.856,A 0.000,B 0.000,C 90.000,E1 10.074} C_DIS
LIN {X -0.012,Y -366.300,Z 1446.854,A 0.000,B 0.000,C 90.000,E1 9.726} C_DIS
LIN {X -0.133,Y -361.701,Z 1446.821,A 0.000,B 0.000,C 90.000,E1 3.784} C_DIS
LIN {X -0.052,Y -360.908,Z 1446.802,A 0.000,B 0.000,C 90.000,E1 0.401} C_DIS
LIN {X 0.137,Y -360.684,Z 1446.799,A 0.000,B 0.000,C 90.000,E1 359.771} C_DIS
LIN {X -0.053,Y -359.426,Z 1446.770,A 0.000,B 0.000,C 90.000,E1 354.546} C_DIS
LIN {X 0.070,Y -358.890,Z 1446.759,A 0.000,B 0.000,C 90.000,E1 352.648} C_DIS
LIN {X -0.020,Y -359.563,Z 1446.726,A 0.000,B 0.000,C 90.000,E1 346.645} C_DIS
LIN {X 0.001,Y -361.801,Z 1446.684,A 0.000,B 0.000,C 90.000,E1 339.135} C_DIS
LIN {X -0.154,Y -362.053,Z 1446.680,A 0.000,B 0.000,C 90.000,E1 338.411} C_DIS
LIN {X 0.189,Y -365.980,Z 1446.643,A 0.000,B 0.000,C 90.000,E1 331.641} C_DIS
LIN {X 0.029,Y -366.387,Z 1446.639,A 0.000,B 0.000,C 90.000,E1 330.923} C_DIS
LIN {X -0.031,Y -371.355,Z 1446.604,A 0.000,B 0.000,C 90.000,E1 324.642} C_DIS
LIN {X -0.043,Y -371.766,Z 1446.602,A 0.000,B 0.000,C 90.000,E1 324.276} C_DIS
LIN {X 0.013,Y -377.358,Z 1446.567,A 0.000,B 0.000,C 90.000,E1 318.038} C_DIS
LIN {X 0.012,Y -378.235,Z 1446.563,A 0.000,B 0.000,C 90.000,E1 317.310} C_DIS
LIN {X 0.002,Y -383.940,Z 1446.531,A 0.000,B 0.000,C 90.000,E1 311.515} C_DIS
LIN {X 0.088,Y -384.893,Z 1446.527,A 0.000,B 0.000,C 90.000,E1 310.782} C_DIS
LIN {X 0.262,Y -390.610,Z 1446.495,A 0.000,B 0.000,C 90.000,E1 305.025} C_DIS
LIN {X 0.106,Y -391.104,Z 1446.493,A 0.000,B 0.000,C 90.000,E1 304.692} C_DIS
LIN {X 0.022,Y -391.648,Z 1446.489,A 0.000,B 0.000,C 90.000,E1 303.992} C_DIS
LIN {X -0.080,Y -396.825,Z 1446.459,A 0.000,B 0.000,C 90.000,E1 298.693} C_DIS
LIN {X -0.210,Y -397.120,Z 1446.457,A 0.000,B 0.000,C 90.000,E1 298.359} C_DIS
LIN {X -0.055,Y -401.597,Z 1446.426,A 0.000,B 0.000,C 90.000,E1 292.717} C_DIS
LIN {X 0.222,Y -404.659,Z 1446.395,A 0.000,B 0.000,C 90.000,E1 287.094} C_DIS
LIN {X -0.079,Y -404.735,Z 1446.391,A 0.000,B 0.000,C 90.000,E1 286.441} C_DIS
LIN {X 0.214,Y -406.099,Z 1446.364,A 0.000,B 0.000,C 90.000,E1 281.535} C_DIS
LIN {X -0.176,Y -406.094,Z 1446.362,A 0.000,B 0.000,C 90.000,E1 281.243} C_DIS
LIN {X -0.097,Y -405.680,Z 1446.333,A 0.000,B 0.000,C 90.000,E1 276.024} C_DIS
LIN {X -0.165,Y -405.058,Z 1446.328,A 0.000,B 0.000,C 90.000,E1 274.992} C_DIS
LIN {X -0.060,Y -403.497,Z 1446.304,A 0.000,B 0.000,C 90.000,E1 270.802} C_DIS
LIN {X -0.092,Y -403.288,Z 1446.302,A 0.000,B 0.000,C 90.000,E1 270.458} C_DIS
LIN {X 0.091,Y -398.931,Z 1446.271,A 0.000,B 0.000,C 90.000,E1 264.837} C_DIS
LIN {X -0.040,Y -393.108,Z 1446.242,A 0.000,B 0.000,C 90.000,E1 259.567} C_DIS
LIN {X -0.079,Y -392.835,Z 1446.240,A 0.000,B 0.000,C 90.000,E1 259.218} C_DIS
LIN {X 0.034,Y -385.993,Z 1446.212,A 0.000,B 0.000,C 90.000,E1 254.212} C_DIS
LIN {X -0.026,Y -385.267,Z 1446.208,A 0.000,B 0.000,C 90.000,E1 253.504} C_DIS
LIN {X -0.004,Y -384.768,Z 1446.206,A 0.000,B 0.000,C 90.000,E1 253.142} C_DIS
LIN {X 0.221,Y -377.973,Z 1446.182,A 0.000,B 0.000,C 90.000,E1 248.773} C_DIS
LIN {X -0.044,Y -376.233,Z 1446.174,A 0.000,B 0.000,C 90.000,E1 247.358} C_DIS
LIN {X 0.057,Y -374.944,Z 1446.170,A 0.000,B 0.000,C 90.000,E1 246.613} C_DIS
LIN {X -0.208,Y -368.417,Z 1446.148,A 0.000,B 0.000,C 90.000,E1 242.615} C_DIS
LIN {X 0.097,Y -366.047,Z 1446.137,A 0.000,B 0.000,C 90.000,E1 240.717} C_DIS
LIN {X 0.004,Y -359.196,Z 1446.115,A 0.000,B 0.000,C 90.000,E1 236.628} C_DIS
LIN {X 0.021,Y -355.842,Z 1446.100,A 0.000,B 0.000,C 90.000,E1 233.989} C_DIS
LIN {X -0.173,Y -348.793,Z 1446.075,A 0.000,B 0.000,C 90.000,E1 229.461} C_DIS
LIN {X -0.097,Y -346.185,Z 1446.062,A 0.000,B 0.000,C 90.000,E1 227.148} C_DIS
LIN {X -0.088,Y -345.065,Z 1446.058,A 0.000,B 0.000,C 90.000,E1 226.377} C_DIS
LIN {X 0.094,Y -338.586,Z 1446.030,A 0.000,B 0.000,C 90.000,E1 221.310} C_DIS
LIN {X 0.094,Y -336.840,Z 1446.019,A 0.000,B 0.000,C 90.000,E1 219.358} C_DIS
LIN {X 0.014,Y -330.861,Z 1445.988,A 0.000,B 0.000,C 90.000,E1 213.865} C_DIS
LIN {X 0.149,Y -329.296,Z 1445.975,A 0.000,B 0.000,C 90.000,E1 211.465} C_DIS
LIN {X -0.154,Y -324.669,Z 1445.942,A 0.000,B 0.000,C 90.000,E1 205.540} C_DIS
LIN {X 0.174,Y -323.837,Z 1445.928,A 0.000,B 0.000,C 90.000,E1 203.078} C_DIS
LIN {X -0.017,Y -321.124,Z 1445.881,A 0.000,B 0.000,C 90.000,E1 194.662} C_DIS
LIN {X 0.138,Y -320.932,Z 1445.877,A 0.000,B 0.000,C 90.000,E1 193.828} C_DIS
LIN {X -0.076,Y -321.562,Z 1445.832,A 0.000,B 0.000,C 90.000,E1 185.796} C_DIS
LIN {X -0.143,Y -324.415,Z 1445.790,A 0.000,B 0.000,C 90.000,E1 178.165} C_DIS
LIN {X -0.141,Y -325.376,Z 1445.783,A 0.000,B 0.000,C 90.000,E1 176.963} C_DIS
LIN {X -0.100,Y -329.112,Z 1445.750,A 0.000,B 0.000,C 90.000,E1 170.971} C_DIS
LIN {X 0.061,Y -334.260,Z 1445.726,A 0.000,B 0.000,C 90.000,E1 166.589} C_DIS
LIN {X 0.067,Y -335.488,Z 1445.719,A 0.000,B 0.000,C 90.000,E1 165.408} C_DIS
LIN {X 0.146,Y -338.378,Z 1445.705,A 0.000,B 0.000,C 90.000,E1 162.906} C_DIS
LIN {X 0.135,Y -395.108,Z 1445.705,A 0.000,B 0.000,C 90.000,E1 162.906} C_DIS
LIN {X 0.129,Y -398.171,Z 1445.705,A 0.000,B 0.000,C 90.000,E1 162.851} C_DIS
LIN {X -0.142,Y -399.822,Z 1445.705,A 0.000,B 0.000,C 90.000,E1 162.834} C_DIS
LIN {X 0.052,Y -402.964,Z 1445.704,A 0.000,B 0.000,C 90.000,E1 162.670} C_DIS
LIN {X -0.138,Y -405.904,Z 1445.703,A 0.000,B 0.000,C 90.000,E1 162.543} C_DIS
LIN {X 0.081,Y -411.998,Z 1445.701,A 0.000,B 0.000,C 90.000,E1 162.127} C_DIS
LIN {X -0.149,Y -416.656,Z 1445.699,A 0.000,B 0.000,C 90.000,E1 161.819} C_DIS
LIN {X 0.172,Y -422.827,Z 1445.696,A 0.000,B 0.000,C 90.000,E1 161.275} C_DIS
LIN {X 0.064,Y -436.452,Z 1445.690,A 0.000,B 0.000,C 90.000,E1 160.115} C_DIS
LIN {X -0.012,Y -448.764,Z 1445.684,A 0.000,B 0.000,C 90.000,E1 159.082} C_DIS
LIN {X 0.073,Y -462.441,Z 1445.677,A 0.000,B 0.000,C 90.000,E1 157.922} C_DIS
LIN {X -0.139,Y -472.966,Z 1445.672,A 0.000,B 0.000,C 90.000,E1 157.050} C_DIS
LIN {X 0.189,Y -483.348,Z 1445.667,A 0.000,B 0.000,C 90.000,E1 156.102} C_DIS
LIN {X 0.124,Y -493.393,Z 1445.662,A 0.000,B 0.000,C 90.000,E1 155.177} C_DIS
LIN {X -0.201,Y -500.251,Z 1445.658,A 0.000,B 0.000,C 90.000,E1 154.537} C_DIS
LIN {X 0.038,Y -505.606,Z 1445.655,A 0.000,B 0.000,C 90.000,E1 153.948} C_DIS
LIN {X 0.086,Y -509.499,Z 1445.653,A 0.000,B 0.000,C 90.000,E1 153.512} C_DIS
LIN {X -0.048,Y -515.467,Z 1445.649,A 0.000,B 0.000,C 90.000,E1 152.794} C_DIS
LIN {X -0.106,Y -518.803,Z 1445.646,A 0.000,B 0.000,C 90.000,E1 152.359} C_DIS
LIN {X -0.069,Y -522.771,Z 1445.643,A 0.000,B 0.000,C 90.000,E1 151.769} C_DIS
LIN {X -0.156,Y -527.086,Z 1445.639,A 0.000,B 0.000,C 90.000,E1 151.051} C_DIS
LIN {X 0.097,Y -529.467,Z 1445.637,A 0.000,B 0.000,C 90.000,E1 150.589} C_DIS
LIN {X 0.069,Y -532.915,Z 1445.633,A 0.000,B 0.000,C 90.000,E1 149.871} C_DIS
LIN {X 0.066,Y -535.998,Z 1445.629,A 0.000,B 0.000,C 90.000,E1 149.154} C_DIS
LIN {X 0.045,Y -538.189,Z 1445.625,A 0.000,B 0.000,C 90.000,E1 148.584} C_DIS
LIN {X -0.058,Y -541.138,Z 1445.621,A 0.000,B 0.000,C 90.000,E1 147.740} C_DIS
LIN {X -0.030,Y -542.884,Z 1445.618,A 0.000,B 0.000,C 90.000,E1 147.168} C_DIS
LIN {X 0.234,Y -546.008,Z 1445.611,A 0.000,B 0.000,C 90.000,E1 146.008} C_DIS
LIN {X 0.043,Y -548.089,Z 1445.607,A 0.000,B 0.000,C 90.000,E1 145.182} C_DIS
LIN {X 0.137,Y -549.389,Z 1445.604,A 0.000,B 0.000,C 90.000,E1 144.609} C_DIS
LIN {X 0.033,Y -551.512,Z 1445.597,A 0.000,B 0.000,C 90.000,E1 143.497} C_DIS
LIN {X 0.216,Y -552.838,Z 1445.593,A 0.000,B 0.000,C 90.000,E1 142.637} C_DIS
LIN {X 0.046,Y -554.414,Z 1445.586,A 0.000,B 0.000,C 90.000,E1 141.537} C_DIS
LIN {X -0.101,Y -555.647,Z 1445.580,A 0.000,B 0.000,C 90.000,E1 140.436} C_DIS
LIN {X 0.125,Y -556.740,Z 1445.574,A 0.000,B 0.000,C 90.000,E1 139.299} C_DIS
LIN {X 0.027,Y -557.936,Z 1445.566,A 0.000,B 0.000,C 90.000,E1 137.919} C_DIS
LIN {X -0.056,Y -558.980,Z 1445.559,A 0.000,B 0.000,C 90.000,E1 136.539} C_DIS
LIN {X 0.189,Y -559.731,Z 1445.552,A 0.000,B 0.000,C 90.000,E1 135.405} C_DIS
LIN {X -0.346,Y -560.276,Z 1445.546,A 0.000,B 0.000,C 90.000,E1 134.352} C_DIS
LIN {X -0.084,Y -560.714,Z 1445.540,A 0.000,B 0.000,C 90.000,E1 133.218} C_DIS
LIN {X 0.126,Y -560.981,Z 1445.536,A 0.000,B 0.000,C 90.000,E1 132.366} C_DIS
LIN {X -0.034,Y -561.141,Z 1445.531,A 0.000,B 0.000,C 90.000,E1 131.553} C_DIS
LIN {X -0.206,Y -561.223,Z 1445.519,A 0.000,B 0.000,C 90.000,E1 129.358} C_DIS
LIN {X 0.187,Y -561.243,Z 1445.511,A 0.000,B 0.000,C 90.000,E1 127.935} C_DIS
LIN {X -0.114,Y -561.218,Z 1445.503,A 0.000,B 0.000,C 90.000,E1 126.583} C_DIS
LIN {X 0.045,Y -561.039,Z 1445.496,A 0.000,B 0.000,C 90.000,E1 125.185} C_DIS
LIN {X 0.203,Y -560.755,Z 1445.488,A 0.000,B 0.000,C 90.000,E1 123.785} C_DIS
LIN {X 0.041,Y -560.467,Z 1445.480,A 0.000,B 0.000,C 90.000,E1 122.418} C_DIS
LIN {X 0.219,Y -560.332,Z 1445.469,A 0.000,B 0.000,C 90.000,E1 120.463} C_DIS
LIN {X -0.014,Y -560.823,Z 1445.454,A 0.000,B 0.000,C 90.000,E1 117.719} C_DIS
LIN {X 0.049,Y -561.325,Z 1445.445,A 0.000,B 0.000,C 90.000,E1 116.052} C_DIS
LIN {X 0.115,Y -561.871,Z 1445.436,A 0.000,B 0.000,C 90.000,E1 114.387} C_DIS
LIN {X -0.078,Y -562.318,Z 1445.428,A 0.000,B 0.000,C 90.000,E1 113.025} C_DIS
LIN {X 0.068,Y -562.912,Z 1445.419,A 0.000,B 0.000,C 90.000,E1 111.354} C_DIS
LIN {X 0.132,Y -563.918,Z 1445.406,A 0.000,B 0.000,C 90.000,E1 109.141} C_DIS
LIN {X -0.265,Y -564.056,Z 1445.405,A 0.000,B 0.000,C 90.000,E1 108.906} C_DIS
LIN {X 0.180,Y -565.228,Z 1445.400,A 0.000,B 0.000,C 90.000,E1 108.000} C_DIS
LIN {X 0.129,Y -566.389,Z 1445.399,A 0.000,B 0.000,C 90.000,E1 107.764} C_DIS
LIN {X -0.085,Y -567.296,Z 1445.397,A 0.000,B 0.000,C 90.000,E1 107.511} C_DIS
LIN {X 0.032,Y -569.450,Z 1445.396,A 0.000,B 0.000,C 90.000,E1 107.221} C_DIS
LIN {X -0.083,Y -575.662,Z 1445.393,A 0.000,B 0.000,C 90.000,E1 106.677} C_DIS
LIN {X 0.266,Y -579.665,Z 1445.391,A 0.000,B 0.000,C 90.000,E1 106.315} C_DIS
LIN {X 0.135,Y -584.974,Z 1445.388,A 0.000,B 0.000,C 90.000,E1 105.843} C_DIS
LIN {X 0.087,Y -589.781,Z 1445.385,A 0.000,B 0.000,C 90.000,E1 105.190} C_DIS
LIN {X 0.006,Y -590.592,Z 1445.384,A 0.000,B 0.000,C 90.000,E1 105.064} C_DIS
LIN {X -0.126,Y -593.230,Z 1445.380,A 0.000,B 0.000,C 90.000,E1 104.411} C_DIS
LIN {X 0.142,Y -594.018,Z 1445.379,A 0.000,B 0.000,C 90.000,E1 104.120} C_DIS
LIN {X 0.116,Y -594.995,Z 1445.376,A 0.000,B 0.000,C 90.000,E1 103.592} C_DIS
LIN {X 0.090,Y -596.244,Z 1445.370,A 0.000,B 0.000,C 90.000,E1 102.535} C_DIS
LIN {X -0.205,Y -596.453,Z 1445.368,A 0.000,B 0.000,C 90.000,E1 102.299} C_DIS
LIN {X -0.210,Y -596.516,Z 1445.365,A 0.000,B 0.000,C 90.000,E1 101.771} C_DIS
LIN {X -0.216,Y -596.333,Z 1445.362,A 0.000,B 0.000,C 90.000,E1 101.243} C_DIS
LIN {X -0.224,Y -595.662,Z 1445.359,A 0.000,B 0.000,C 90.000,E1 100.715} C_DIS
LIN {X -0.046,Y -595.192,Z 1445.358,A 0.000,B 0.000,C 90.000,E1 100.433} C_DIS
LIN {X -0.060,Y -593.836,Z 1445.355,A 0.000,B 0.000,C 90.000,E1 99.905} C_DIS
LIN {X -0.087,Y -592.218,Z 1445.352,A 0.000,B 0.000,C 90.000,E1 99.378} C_DIS
LIN {X -0.222,Y -590.201,Z 1445.349,A 0.000,B 0.000,C 90.000,E1 98.859} C_DIS
LIN {X 0.043,Y -588.863,Z 1445.348,A 0.000,B 0.000,C 90.000,E1 98.568} C_DIS
LIN {X 0.094,Y -586.636,Z 1445.345,A 0.000,B 0.000,C 90.000,E1 98.163} C_DIS
LIN {X -0.053,Y -580.514,Z 1445.340,A 0.000,B 0.000,C 90.000,E1 97.239} C_DIS
LIN {X -0.259,Y -576.639,Z 1445.337,A 0.000,B 0.000,C 90.000,E1 96.720} C_DIS
LIN {X -0.053,Y -574.587,Z 1445.336,A 0.000,B 0.000,C 90.000,E1 96.429} C_DIS
LIN {X 0.275,Y -573.437,Z 1445.335,A 0.000,B 0.000,C 90.000,E1 96.201} C_DIS
LIN {X 0.274,Y -570.261,Z 1445.330,A 0.000,B 0.000,C 90.000,E1 95.391} C_DIS
LIN {X 0.216,Y -569.903,Z 1445.328,A 0.000,B 0.000,C 90.000,E1 95.049} C_DIS
LIN {X 0.291,Y -569.740,Z 1445.326,A 0.000,B 0.000,C 90.000,E1 94.588} C_DIS
LIN {X -0.032,Y -570.489,Z 1445.317,A 0.000,B 0.000,C 90.000,E1 92.980} C_DIS
LIN {X 0.070,Y -571.603,Z 1445.309,A 0.000,B 0.000,C 90.000,E1 91.604} C_DIS
LIN {X -0.112,Y -573.279,Z 1445.298,A 0.000,B 0.000,C 90.000,E1 89.714} C_DIS
LIN {X -0.237,Y -574.970,Z 1445.288,A 0.000,B 0.000,C 90.000,E1 87.822} C_DIS
LIN {X -0.144,Y -576.946,Z 1445.276,A 0.000,B 0.000,C 90.000,E1 85.641} C_DIS
LIN {X 0.243,Y -579.215,Z 1445.262,A 0.000,B 0.000,C 90.000,E1 83.166} C_DIS
LIN {X 0.036,Y -581.328,Z 1445.250,A 0.000,B 0.000,C 90.000,E1 81.027} C_DIS
LIN {X 0.075,Y -583.442,Z 1445.238,A 0.000,B 0.000,C 90.000,E1 78.870} C_DIS
LIN {X 0.135,Y -584.807,Z 1445.231,A 0.000,B 0.000,C 90.000,E1 77.521} C_DIS
LIN {X 0.136,Y -586.300,Z 1445.220,A 0.000,B 0.000,C 90.000,E1 75.644} C_DIS
LIN {X -0.192,Y -587.235,Z 1445.213,A 0.000,B 0.000,C 90.000,E1 74.338} C_DIS
LIN {X -0.003,Y -588.504,Z 1445.201,A 0.000,B 0.000,C 90.000,E1 72.181} C_DIS
LIN {X -0.156,Y -589.587,Z 1445.189,A 0.000,B 0.000,C 90.000,E1 70.061} C_DIS
LIN {X -0.086,Y -590.744,Z 1445.177,A 0.000,B 0.000,C 90.000,E1 67.922} C_DIS
LIN {X 0.122,Y -591.659,Z 1445.168,A 0.000,B 0.000,C 90.000,E1 66.305} C_DIS
LIN {X 0.106,Y -593.694,Z 1445.152,A 0.000,B 0.000,C 90.000,E1 63.384} C_DIS
LIN {X 0.261,Y -595.002,Z 1445.142,A 0.000,B 0.000,C 90.000,E1 61.513} C_DIS
LIN {X 0.210,Y -596.581,Z 1445.132,A 0.000,B 0.000,C 90.000,E1 59.665} C_DIS
LIN {X -0.227,Y -598.003,Z 1445.123,A 0.000,B 0.000,C 90.000,E1 58.122} C_DIS
LIN {X 0.046,Y -598.916,Z 1445.117,A 0.000,B 0.000,C 90.000,E1 57.041} C_DIS
LIN {X 0.067,Y -600.111,Z 1445.110,A 0.000,B 0.000,C 90.000,E1 55.722} C_DIS
LIN {X 0.111,Y -601.297,Z 1445.102,A 0.000,B 0.000,C 90.000,E1 54.402} C_DIS
LIN {X -0.069,Y -602.429,Z 1445.094,A 0.000,B 0.000,C 90.000,E1 52.844} C_DIS
LIN {X -0.122,Y -603.345,Z 1445.086,A 0.000,B 0.000,C 90.000,E1 51.537} C_DIS
LIN {X -0.035,Y -603.957,Z 1445.080,A 0.000,B 0.000,C 90.000,E1 50.481} C_DIS
LIN {X -0.120,Y -604.385,Z 1445.076,A 0.000,B 0.000,C 90.000,E1 49.703} C_DIS
LIN {X -0.024,Y -604.643,Z 1445.070,A 0.000,B 0.000,C 90.000,E1 48.647} C_DIS
LIN {X 0.131,Y -605.010,Z 1445.059,A 0.000,B 0.000,C 90.000,E1 46.539} C_DIS
LIN {X -0.022,Y -605.040,Z 1445.054,A 0.000,B 0.000,C 90.000,E1 45.769} C_DIS
LIN {X -0.183,Y -604.986,Z 1445.050,A 0.000,B 0.000,C 90.000,E1 45.000} C_DIS
LIN {X 0.088,Y -604.718,Z 1445.046,A 0.000,B 0.000,C 90.000,E1 44.190} C_DIS
LIN {X -0.062,Y -604.317,Z 1445.041,A 0.000,B 0.000,C 90.000,E1 43.419} C_DIS
LIN {X 0.243,Y -603.391,Z 1445.034,A 0.000,B 0.000,C 90.000,E1 42.081} C_DIS
LIN {X -0.122,Y -602.500,Z 1445.028,A 0.000,B 0.000,C 90.000,E1 41.067} C_DIS
LIN {X -0.050,Y -601.386,Z 1445.022,A 0.000,B 0.000,C 90.000,E1 40.011} C_DIS
LIN {X 0.244,Y -599.730,Z 1445.015,A 0.000,B 0.000,C 90.000,E1 38.669} C_DIS
LIN {X -0.106,Y -598.245,Z 1445.009,A 0.000,B 0.000,C 90.000,E1 37.649} C_DIS
LIN {X -0.233,Y -597.002,Z 1445.005,A 0.000,B 0.000,C 90.000,E1 36.870} C_DIS
LIN {X -0.369,Y -595.511,Z 1445.000,A 0.000,B 0.000,C 90.000,E1 36.091} C_DIS
LIN {X 0.309,Y -593.842,Z 1444.996,A 0.000,B 0.000,C 90.000,E1 35.231} C_DIS
LIN {X 0.223,Y -590.666,Z 1444.989,A 0.000,B 0.000,C 90.000,E1 33.913} C_DIS
LIN {X -0.115,Y -587.726,Z 1444.983,A 0.000,B 0.000,C 90.000,E1 32.880} C_DIS
LIN {X -0.179,Y -585.320,Z 1444.978,A 0.000,B 0.000,C 90.000,E1 32.084} C_DIS
LIN {X -0.130,Y -583.560,Z 1444.975,A 0.000,B 0.000,C 90.000,E1 31.544} C_DIS
LIN {X 0.069,Y -580.529,Z 1444.971,A 0.000,B 0.000,C 90.000,E1 30.718} C_DIS
LIN {X 0.005,Y -577.638,Z 1444.967,A 0.000,B 0.000,C 90.000,E1 30.050} C_DIS
LIN {X 0.255,Y -573.176,Z 1444.962,A 0.000,B 0.000,C 90.000,E1 29.077} C_DIS
LIN {X -0.151,Y -569.628,Z 1444.958,A 0.000,B 0.000,C 90.000,E1 28.437} C_DIS
LIN {X 0.186,Y -565.829,Z 1444.954,A 0.000,B 0.000,C 90.000,E1 27.719} C_DIS
LIN {X 0.287,Y -560.178,Z 1444.949,A 0.000,B 0.000,C 90.000,E1 26.744} C_DIS
LIN {X 0.174,Y -554.932,Z 1444.944,A 0.000,B 0.000,C 90.000,E1 25.924} C_DIS
LIN {X 0.127,Y -550.196,Z 1444.940,A 0.000,B 0.000,C 90.000,E1 25.232} C_DIS
LIN {X 0.142,Y -543.925,Z 1444.936,A 0.000,B 0.000,C 90.000,E1 24.387} C_DIS
LIN {X 0.125,Y -539.425,Z 1444.932,A 0.000,B 0.000,C 90.000,E1 23.823} C_DIS
LIN {X -0.065,Y -533.478,Z 1444.928,A 0.000,B 0.000,C 90.000,E1 23.131} C_DIS
LIN {X 0.181,Y -527.263,Z 1444.925,A 0.000,B 0.000,C 90.000,E1 22.386} C_DIS
LIN {X 0.038,Y -518.305,Z 1444.919,A 0.000,B 0.000,C 90.000,E1 21.408} C_DIS
LIN {X 0.090,Y -509.178,Z 1444.914,A 0.000,B 0.000,C 90.000,E1 20.429} C_DIS
LIN {X 0.184,Y -498.567,Z 1444.907,A 0.000,B 0.000,C 90.000,E1 19.322} C_DIS
LIN {X -0.078,Y -479.694,Z 1444.897,A 0.000,B 0.000,C 90.000,E1 17.402} C_DIS
LIN {X -0.161,Y -470.201,Z 1444.891,A 0.000,B 0.000,C 90.000,E1 16.386} C_DIS
LIN {X 0.202,Y -465.858,Z 1444.889,A 0.000,B 0.000,C 90.000,E1 15.898} C_DIS
LIN {X 0.173,Y -461.279,Z 1444.886,A 0.000,B 0.000,C 90.000,E1 15.481} C_DIS
LIN {X -0.175,Y -456.295,Z 1444.884,A 0.000,B 0.000,C 90.000,E1 15.134} C_DIS
LIN {X -0.159,Y -452.616,Z 1444.883,A 0.000,B 0.000,C 90.000,E1 14.898} C_DIS
LIN {X -0.106,Y -450.114,Z 1444.882,A 0.000,B 0.000,C 90.000,E1 14.773} C_DIS
LIN {X -0.037,Y -448.605,Z 1444.882,A 0.000,B 0.000,C 90.000,E1 14.717} C_DIS
LIN {X -0.152,Y -447.710,Z 1444.882,A 0.000,B 0.000,C 90.000,E1 14.717} C_DIS
LIN {X -0.158,Y -370.195,Z 1444.882,A 0.000,B 0.000,C 90.000,E1 14.717} C_DIS
LIN {X 0.181,Y -366.548,Z 1444.856,A 0.000,B 0.000,C 90.000,E1 10.018} C_DIS
LIN {X -0.106,Y -365.838,Z 1444.852,A 0.000,B 0.000,C 90.000,E1 9.321} C_DIS
LIN {X -0.092,Y -361.397,Z 1444.817,A 0.000,B 0.000,C 90.000,E1 2.980} C_DIS
LIN {X -0.001,Y -360.906,Z 1444.802,A 0.000,B 0.000,C 90.000,E1 0.344} C_DIS
LIN {X 0.105,Y -360.314,Z 1444.795,A 0.000,B 0.000,C 90.000,E1 359.026} C_DIS
LIN {X -0.053,Y -359.426,Z 1444.770,A 0.000,B 0.000,C 90.000,E1 354.546} C_DIS
LIN {X 0.070,Y -358.890,Z 1444.759,A 0.000,B 0.000,C 90.000,E1 352.648} C_DIS
LIN {X -0.020,Y -359.563,Z 1444.726,A 0.000,B 0.000,C 90.000,E1 346.645} C_DIS
LIN {X 0.001,Y -361.801,Z 1444.684,A 0.000,B 0.000,C 90.000,E1 339.135} C_DIS
LIN {X -0.154,Y -362.053,Z 1444.680,A 0.000,B 0.000,C 90.000,E1 338.411} C_DIS
LIN {X 0.189,Y -365.980,Z 1444.643,A 0.000,B 0.000,C 90.000,E1 331.641} C_DIS
LIN {X 0.029,Y -366.387,Z 1444.639,A 0.000,B 0.000,C 90.000,E1 330.923} C_DIS
LIN {X -0.031,Y -371.355,Z 1444.604,A 0.000,B 0.000,C 90.000,E1 324.642} C_DIS
LIN {X -0.043,Y -371.766,Z 1444.602,A 0.000,B 0.000,C 90.000,E1 324.276} C_DIS
LIN {X 0.013,Y -377.358,Z 1444.567,A 0.000,B 0.000,C 90.000,E1 318.038} C_DIS
LIN {X 0.012,Y -378.235,Z 1444.563,A 0.000,B 0.000,C 90.000,E1 317.310} C_DIS
LIN {X 0.002,Y -383.940,Z 1444.531,A 0.000,B 0.000,C 90.000,E1 311.515} C_DIS
LIN {X 0.088,Y -384.893,Z 1444.527,A 0.000,B 0.000,C 90.000,E1 310.782} C_DIS
LIN {X 0.262,Y -390.610,Z 1444.495,A 0.000,B 0.000,C 90.000,E1 305.025} C_DIS
LIN {X 0.106,Y -391.104,Z 1444.493,A 0.000,B 0.000,C 90.000,E1 304.692} C_DIS
LIN {X 0.022,Y -391.648,Z 1444.489,A 0.000,B 0.000,C 90.000,E1 303.992} C_DIS
LIN {X -0.080,Y -396.825,Z 1444.459,A 0.000,B 0.000,C 90.000,E1 298.693} C_DIS
LIN {X -0.210,Y -397.120,Z 1444.457,A 0.000,B 0.000,C 90.000,E1 298.359} C_DIS
LIN {X -0.055,Y -401.597,Z 1444.426,A 0.000,B 0.000,C 90.000,E1 292.717} C_DIS
LIN {X 0.222,Y -404.659,Z 1444.395,A 0.000,B 0.000,C 90.000,E1 287.094} C_DIS
LIN {X -0.079,Y -404.735,Z 1444.391,A 0.000,B 0.000,C 90.000,E1 286.441} C_DIS
LIN {X 0.214,Y -406.099,Z 1444.364,A 0.000,B 0.000,C 90.000,E1 281.535} C_DIS
LIN {X -0.176,Y -406.094,Z 1444.362,A 0.000,B 0.000,C 90.000,E1 281.243} C_DIS
LIN {X -0.097,Y -405.680,Z 1444.333,A 0.000,B 0.000,C 90.000,E1 276.024} C_DIS
LIN {X -0.165,Y -405.058,Z 1444.328,A 0.000,B 0.000,C 90.000,E1 274.992} C_DIS
LIN {X -0.060,Y -403.497,Z 1444.304,A 0.000,B 0.000,C 90.000,E1 270.802} C_DIS
LIN {X -0.092,Y -403.288,Z 1444.302,A 0.000,B 0.000,C 90.000,E1 270.458} C_DIS
LIN {X 0.091,Y -398.931,Z 1444.271,A 0.000,B 0.000,C 90.000,E1 264.837} C_DIS
LIN {X -0.040,Y -393.108,Z 1444.242,A 0.000,B 0.000,C 90.000,E1 259.567} C_DIS
LIN {X -0.079,Y -392.835,Z 1444.240,A 0.000,B 0.000,C 90.000,E1 259.218} C_DIS
LIN {X 0.034,Y -385.993,Z 1444.212,A 0.000,B 0.000,C 90.000,E1 254.212} C_DIS
LIN {X -0.026,Y -385.267,Z 1444.208,A 0.000,B 0.000,C 90.000,E1 253.504} C_DIS
LIN {X -0.004,Y -384.768,Z 1444.206,A 0.000,B 0.000,C 90.000,E1 253.142} C_DIS
LIN {X 0.221,Y -377.973,Z 1444.182,A 0.000,B 0.000,C 90.000,E1 248.773} C_DIS
LIN {X -0.044,Y -376.233,Z 1444.174,A 0.000,B 0.000,C 90.000,E1 247.358} C_DIS
LIN {X 0.057,Y -374.944,Z 1444.170,A 0.000,B 0.000,C 90.000,E1 246.613} C_DIS
LIN {X -0.208,Y -368.417,Z 1444.148,A 0.000,B 0.000,C 90.000,E1 242.615} C_DIS
LIN {X 0.097,Y -366.047,Z 1444.137,A 0.000,B 0.000,C 90.000,E1 240.717} C_DIS
LIN {X 0.004,Y -359.196,Z 1444.115,A 0.000,B 0.000,C 90.000,E1 236.628} C_DIS
LIN {X 0.021,Y -355.842,Z 1444.100,A 0.000,B 0.000,C 90.000,E1 233.989} C_DIS
LIN {X -0.173,Y -348.793,Z 1444.075,A 0.000,B 0.000,C 90.000,E1 229.461} C_DIS
LIN {X -0.097,Y -346.185,Z 1444.062,A 0.000,B 0.000,C 90.000,E1 227.148} C_DIS
LIN {X -0.088,Y -345.065,Z 1444.058,A 0.000,B 0.000,C 90.000,E1 226.377} C_DIS
LIN {X 0.094,Y -338.586,Z 1444.030,A 0.000,B 0.000,C 90.000,E1 221.310} C_DIS
LIN {X 0.094,Y -336.840,Z 1444.019,A 0.000,B 0.000,C 90.000,E1 219.358} C_DIS
LIN {X 0.014,Y -330.861,Z 1443.988,A 0.000,B 0.000,C 90.000,E1 213.865} C_DIS
LIN {X 0.149,Y -329.296,Z 1443.975,A 0.000,B 0.000,C 90.000,E1 211.465} C_DIS
LIN {X -0.154,Y -324.669,Z 1443.942,A 0.000,B 0.000,C 90.000,E1 205.540} C_DIS
LIN {X 0.174,Y -323.837,Z 1443.928,A 0.000,B 0.000,C 90.000,E1 203.078} C_DIS
LIN {X -0.017,Y -321.124,Z 1443.881,A 0.000,B 0.000,C 90.000,E1 194.662} C_DIS
LIN {X 0.138,Y -320.932,Z 1443.877,A 0.000,B 0.000,C 90.000,E1 193.828} C_DIS
LIN {X -0.076,Y -321.562,Z 1443.832,A 0.000,B 0.000,C 90.000,E1 185.796} C_DIS
LIN {X -0.143,Y -324.415,Z 1443.790,A 0.000,B 0.000,C 90.000,E1 178.165} C_DIS
LIN {X -0.141,Y -325.376,Z 1443.783,A 0.000,B 0.000,C 90.000,E1 176.963} C_DIS
LIN {X -0.100,Y -329.112,Z 1443.750,A 0.000,B 0.000,C 90.000,E1 170.971} C_DIS
LIN {X 0.061,Y -334.260,Z 1443.726,A 0.000,B 0.000,C 90.000,E1 166.589} C_DIS
LIN {X 0.067,Y -335.488,Z 1443.719,A 0.000,B 0.000,C 90.000,E1 165.408} C_DIS
LIN {X -0.010,Y -337.516,Z 1443.709,A 0.000,B 0.000,C 90.000,E1 163.614} C_DIS
